// TwinCAT 3 PLC project Imbad160702PLCProgram
// ProgramVersion: 3.1.4020.4
// libraries:
//   Tc2_SerialCom, * (Beckhoff Automation GmbH)
//   Tc2_Standard, * (Beckhoff Automation GmbH)
//   Tc2_System, * (Beckhoff Automation GmbH)
//   Tc2_TcpIp, * (Beckhoff Automation GmbH)
//   Tc2_Utilities, * (Beckhoff Automation GmbH)
//   Tc3_Module, * (Beckhoff Automation GmbH)
//   Tc2_EthernetIP,newest,Beckhoff Automation GmbH
// project tree:
//   DUTs/CycleStationControl/ eAutoBaggerState.TcDUT, eCapInsertStaState.TcDUT, eGoodULStaState.TcDUT, eGoodULNewStaState.TcDUT, eVisionStaState.TcDUT, eOB_StopBeforeVisionState.TcDUT, eRejectStaState.TcDUT, ePistonInsertStaState.TcDUT, eIB_StopRobotClearStaState.TcDUT, eLoadSta1State.TcDUT, eOB_StopRobotClearStaState.TcDUT, eLoadSta2State.TcDUT, eLoadSta3State.TcDUT, eLoadSta4State.TcDUT, ePrimeMoverState.TcDUT, eCycleControlState.TcDUT, OverallStationStatus.TcDUT
//   DUTs/FrameworkDUTs/ ST_EventData.TcDUT
//   DUTs/LotDataDUTs/ eBarrelType.TcDUT, eVisionEnableState.TcDUT, LotDataType.TcDUT, StatusCounts.TcDUT
//   DUTs/Magnemotion/ eMM_HLCStatus.TcDUT, eMM_ResetCmdStatus.TcDUT, eMM_StartupCmdStatus.TcDUT, eMM_VehicleState.TcDUT, eMM_VehMoveToPosCmdStatus.TcDUT, ST_B1Cmd.TcDUT, ST_B1Res.TcDUT, ST_B2Cmd.TcDUT, ST_B2Res.TcDUT, ST_B3Cmd.TcDUT, ST_B3Res.TcDUT, ST_B4Cmd.TcDUT, ST_B4Res.TcDUT, ST_B5Cmd.TcDUT, ST_B8Cmd.TcDUT, ST_B8Res.TcDUT, ST_MM_Header.TcDUT, ST_MM_ResDataNamed.TcDUT, ST_MM_ResHeader.TcDUT, ST_MM_RxFrame.TcDUT, ST_MM_TxFrame.TcDUT, ST_ResD0.TcDUT, ST_ResD1.TcDUT, ST_ResD2.TcDUT, ST_ResD3.TcDUT, ST_ResD4.TcDUT, ST_ResD5.TcDUT, ST_ResD7.TcDUT, ST_VehicleStatus.TcDUT, ST_VehicleStatusHMI.TcDUT, U_MM_CmdData.TcDUT, U_MM_ResCmdDataDetail.TcDUT, U_MM_ResD0CmdDataDetail.TcDUT, U_MM_ResData.TcDUT
//   DUTs/PartsDataDUTs/ ePartStatus.TcDUT, PartDataType.TcDUT, VisionInspectDataType.TcDUT
//   GVLs/ CONFIG.TcGVL, GVL_IO.TcGVL, Logging.TcGVL, LotsData.TcGVL, MM_CONST.TcGVL, PartsData.TcGVL, Stations.TcGVL, STATUS.TcGVL, VIS_CONST.TcGVL
//   / PlcTask.TcTTO, SerialComTask.TcTTO
//   POUs/ AutoBagger.TcPOU, BurnOffStation.TcPOU, CapInsertStation.TcPOU, CapInsertStation_Old.TcPOU, CheckBounds.TcPOU, CycleControl.TcPOU, GoodULStation_2.TcPOU, GoodULStation_3.TcPOU, GoodULStation_4.TcPOU, GoodUnloadStation.TcPOU, IB_StopRobotClearStation.TcPOU, Load1Station.TcPOU, Load2Station.TcPOU, Load3Station.TcPOU, Load4Station.TcPOU, OB_StopRobotClearStation.TcPOU, PistonInsertStation.TcPOU, PrimeMover.TcPOU, MAIN.TcPOU, P_TextModeWrite.TcPOU, P_TextModeWriteLot.TcPOU, RejectStation.TcPOU, GoodULStation_1.TcPOU, RoutePlanner.TcPOU, StationManager.TcPOU, OB_StopBeforeVisionStation.TcPOU, VehicleManager.TcPOU, VisionStation.TcPOU
//   POUs/FrameworkPOUs/ BackgroundEL.TcPOU, EventMsg.TcPOU, EventMsgParams.TcPOU, FB_SerialCom.TcPOU, LotLogging.TcPOU, GetInputsFromFieldBus.TcPOU, MapLockedOutputsfromHMI.TcPOU, PrepareInputsDataStructureForHMI.TcPOU, PrepareOutputsDataStructureForHMI.TcPOU, SetOutputsToFieldBus.TcPOU
//   POUs/MagneMotion/HelperPOUs/ FB_LogFifo.TcPOU, FB_Rx_FrameFifo.TcPOU, FB_Tx_FrameFifo.TcPOU, F_ADSLOGHEXDATA.TcPOU
//   POUs/MagneMotion/ HLCConnection.TcPOU, MMClient.TcPOU, MMStatusMonitor.TcPOU, MM_MsgFormatter.TcPOU, MM_MsgParser.TcPOU
// real-time tasks:
//   TASK PlcTask: cycle T#10ms, priority 20, ADS port 350
//   TASK SerialComTask: cycle T#1ms, priority 16, ADS port 351
// I/O:
//   DEVICE Device 1 (EtherCAT), AmsNetId 5.37.254.56.2.1
//     Term 1 (EK1200) [EK1200-5000 EtherCAT Power supply (2A E-Bus)]
//       Term 2 (EL1809) [EL1809 16Ch. Dig. Input 24V, 3ms]
//       Term 3 (EL1088) [EL1088 8Ch. Dig. Input 24V, 3ms, negative]
//       Term 4 (EL2809) [EL2809 16Ch. Dig. Output 24V, 0.5A]
//       Term 5 (EL3312) [EL3312 2Ch. Ana. Input Thermocouple (TC)]
//       Term 6 (EL4002) [EL4002 2Ch. Ana. Output 0-10V, 12bit]
//       Term 7 (EL6001) [EL6001 Interface (RS232)]
//       Term 20 (EL2624) [EL2624 4Ch. Relay Output, NO (125V AC / 30V DC)]
//       Term 25 (EL2084) [EL2084 4Ch. Dig. Output 24V, 0.5A, switching to negative]
//       Term 10 (EK1122) [EK1122 2 port EtherCAT junction]
//         Box 37 (EP1809-0021) [EP1809-0021 16 Ch. Dig. Input 24V, 3ms, M8]
//         Box 24 (EX260-SEC1) [EX260-SEC1 EtherCAT SI Unit (32DO_PNP) Rev1.2]
//         Box 41 (EP2339-0021) [EP2339-0021 16 Ch. Dig. Input/Output 24V, 0,5A, M8]
//         Box 42 (EP1809-0021) [EP1809-0021 16 Ch. Dig. Input 24V, 3ms, M8]
//         Box 43 (EP1809-0021) [EP1809-0021 16 Ch. Dig. Input 24V, 3ms, M8]
//         Box 11 (EX260-SEC1) [EX260-SEC1 EtherCAT SI Unit (32DO_PNP) Rev1.2]
//         Box 32 (JXCE1) [JXCE1 EtherCAT JXC Rev.1.1]
//   DEVICE Device 2 (TC3 EIP Scanner), AmsNetId 5.55.113.178.3.1
//     CV-X400 Series // <INFO> 192.168.0.31, CV-X400 Series (ProdCode: 5005, Rev: 1.01, Mac: 00:01:fc:21:1c:0d) </INFO> <EDS> </EDS>
// variable links:
//   Imbad160702PLCProgram/Imbad160702PLCProgram Instance <-> Device 1 (EtherCAT)/Term 1 (EK1200)/Term 10 (EK1122)/Box 11 (EX260-SEC1)
//     PlcTask Outputs/GVL_IO.SMCEX260_2_Byte{0..3} <-> Byte {0..3}/Output  (4 links)
//   Imbad160702PLCProgram/Imbad160702PLCProgram Instance <-> Device 1 (EtherCAT)/Term 1 (EK1200)/Term 10 (EK1122)/Box 24 (EX260-SEC1)
//     PlcTask Outputs/GVL_IO.SMCEX260_1_Byte{0..3} <-> Byte {0..3}/Output  (4 links)
//   Imbad160702PLCProgram/Imbad160702PLCProgram Instance <-> Device 1 (EtherCAT)/Term 1 (EK1200)/Term 10 (EK1122)/Box 32 (JXCE1)
//     PlcTask Inputs/GVL_IO.SMC_LEY_XCurrMtrPos <-> Tx PDO1 Mapping/Current position
//     PlcTask Inputs/GVL_IO.SMC_LEY_XUINT0 <-> Tx PDO1 Mapping/Signal allocated to the input port
//     PlcTask Inputs/GVL_IO.SMC_LEY_XUINT1 <-> Tx PDO1 Mapping/Controller information flag
//     PlcTask Outputs/GVL_IO.SMC_LEY_YUINT0 <-> Rx PDO1 Mapping/Output port to which signals are allcated
//   Imbad160702PLCProgram/Imbad160702PLCProgram Instance <-> Device 1 (EtherCAT)/Term 1 (EK1200)/Term 10 (EK1122)/Box 37 (EP1809-0021)
//     PlcTask Inputs/GVL_IO.LD_XPalletCloseExtended_1_2 <-> Channel 2/Input
//     PlcTask Inputs/GVL_IO.LD_XPalletCloseExtended_3_4 <-> Channel 4/Input
//     PlcTask Inputs/GVL_IO.LD_XPalletCloseRetracted_1_2 <-> Channel 1/Input
//     PlcTask Inputs/GVL_IO.LD_XPalletCloseRetracted_3_4 <-> Channel 3/Input
//     PlcTask Inputs/GVL_IO.LD_XPalletHoldDownExtendHome <-> Channel 14/Input
//     PlcTask Inputs/GVL_IO.LD_XPalletHoldRetractEngage <-> Channel 13/Input
//     PlcTask Inputs/GVL_IO.LD_XPalletReleaseExtended <-> Channel 16/Input
//     PlcTask Inputs/GVL_IO.LD_XPalletReleaseHome <-> Channel 15/Input
//     PlcTask Inputs/GVL_IO.PI_XEscapementAtBowl <-> Channel 7/Input
//     PlcTask Inputs/GVL_IO.PI_XEscapementAtInsertLoc <-> Channel 6/Input
//     PlcTask Inputs/GVL_IO.PI_XPalletHoldDownExtended <-> Channel 11/Input
//     PlcTask Inputs/GVL_IO.PI_XPalletHoldDownHome <-> Channel 10/Input
//     PlcTask Inputs/GVL_IO.PI_XPistonPresentEscapement <-> Channel 12/Input
//   Imbad160702PLCProgram/Imbad160702PLCProgram Instance <-> Device 1 (EtherCAT)/Term 1 (EK1200)/Term 10 (EK1122)/Box 41 (EP2339-0021)
//     PlcTask Inputs/GVL_IO.MC_XAirPressureOK <-> Channel 13/Input
//     PlcTask Inputs/GVL_IO.RJ_XPartPresent <-> Channel 16/Input
//     PlcTask Inputs/GVL_IO.UL_1_XBarrelPresent <-> Channel 11/Input
//     PlcTask Inputs/GVL_IO.UL_2_XBarrelPresent <-> Channel 12/Input
//     PlcTask Inputs/GVL_IO.UL_3_XBarrelPresent <-> Channel 14/Input
//     PlcTask Inputs/GVL_IO.UL_4_XBarrelPresent <-> Channel 15/Input
//     PlcTask Inputs/GVL_IO.YU_XLocBit0 <-> Channel 3/Input
//     PlcTask Inputs/GVL_IO.YU_XLocBit1 <-> Channel 4/Input
//     PlcTask Inputs/GVL_IO.YU_XPrepareToLoad <-> Channel 1/Input
//     PlcTask Inputs/GVL_IO.YU_XToolDown <-> Channel 5/Input
//     PlcTask Inputs/GVL_IO.YU_XToolUp <-> Channel 2/Input
//     PlcTask Outputs/GVL_IO.YU_YAckPartsHeld <-> Channel 24/Output
//     PlcTask Outputs/GVL_IO.YU_YIMBADIsOK <-> Channel 22/Output
//     PlcTask Outputs/GVL_IO.YU_YOkToLoad <-> Channel 23/Output
//   Imbad160702PLCProgram/Imbad160702PLCProgram Instance <-> Device 1 (EtherCAT)/Term 1 (EK1200)/Term 10 (EK1122)/Box 42 (EP1809-0021)
//     PlcTask Inputs/GVL_IO.BG_XChute1Closed <-> Channel 14/Input
//     PlcTask Inputs/GVL_IO.BG_XChute2Closed <-> Channel 8/Input
//     PlcTask Inputs/GVL_IO.BG_XChute3Closed <-> Channel 11/Input
//     PlcTask Inputs/GVL_IO.BG_XChute4Closed <-> Channel 12/Input
//     PlcTask Inputs/GVL_IO.BG_XChute1Open <-> Channel 7/Input
//     PlcTask Inputs/GVL_IO.BG_XChute2Open <-> Channel 9/Input
//     PlcTask Inputs/GVL_IO.BG_XChute3Open <-> Channel 10/Input
//     PlcTask Inputs/GVL_IO.BG_XChute4Open <-> Channel 13/Input
//     PlcTask Inputs/GVL_IO.RJ_XPalletHoldDownExtended_Home <-> Channel 4/Input
//     PlcTask Inputs/GVL_IO.RJ_XPalletHoldDownRetracted_Engaged <-> Channel 5/Input
//     PlcTask Inputs/GVL_IO.UL_3_XPalletHoldDownRetracted_Engaged <-> Channel 1/Input
//     PlcTask Inputs/GVL_IO.UL_4_XPalletHoldDownRetracted_Engaged <-> Channel 3/Input
//     PlcTask Inputs/GVL_IO.UL_4_XPalletHoldDownExtended_Home <-> Channel 2/Input
//   Imbad160702PLCProgram/Imbad160702PLCProgram Instance <-> Device 1 (EtherCAT)/Term 1 (EK1200)/Term 10 (EK1122)/Box 43 (EP1809-0021)
//     PlcTask Inputs/GVL_IO.CP_XCapSlideExtended <-> Channel 5/Input
//     PlcTask Inputs/GVL_IO.CP_XCapSlideRetracted <-> Channel 6/Input
//     PlcTask Inputs/GVL_IO.CP_XPalletHoldDownExtended <-> Channel 2/Input
//     PlcTask Inputs/GVL_IO.CP_XPalletHoldDownHome <-> Channel 1/Input
//     PlcTask Inputs/GVL_IO.UL_1_XPalletHoldDownExtended_Home <-> Channel 12/Input
//     PlcTask Inputs/GVL_IO.UL_2_XPalletHoldDownExtended_Home <-> Channel 14/Input
//     PlcTask Inputs/GVL_IO.UL_3_XPalletHoldDownExtended_Home <-> Channel 16/Input
//     PlcTask Inputs/GVL_IO.UL_1_XPalletHoldDownRetracted_Engaged <-> Channel 13/Input
//     PlcTask Inputs/GVL_IO.UL_2_XPalletHoldDownRetracted_Engaged <-> Channel 15/Input
//   Imbad160702PLCProgram/Imbad160702PLCProgram Instance <-> Device 1 (EtherCAT)/Term 1 (EK1200)/Term 2 (EL1809)
//     PlcTask Inputs/GVL_IO.BG_XBaggerOKNoFault <-> Channel 12/Input
//     PlcTask Inputs/GVL_IO.BG_XBaggerReadyForFiller <-> Channel 14/Input
//     PlcTask Inputs/GVL_IO.BG_XBaggerWaitingForLabel <-> Channel 13/Input
//     PlcTask Inputs/GVL_IO.BG_XBagsLow <-> Channel 11/Input
//     PlcTask Inputs/GVL_IO.BU_XAlarm <-> Channel 1/Input
//     PlcTask Inputs/GVL_IO.MC_NotEStopped <-> Channel 7/Input
//     PlcTask Inputs/GVL_IO.MC_XStartPB <-> Channel 3/Input
//     PlcTask Inputs/GVL_IO.MC_XStopPB <-> Channel 4/Input
//   Imbad160702PLCProgram/Imbad160702PLCProgram Instance <-> Device 1 (EtherCAT)/Term 1 (EK1200)/Term 20 (EL2624)
//     PlcTask Outputs/GVL_IO.BG_YFillerTrigger <-> Channel 2/Output
//     PlcTask Outputs/GVL_IO.IZ_YInterrupt <-> Channel 3/Output
//     PlcTask Outputs/GVL_IO.MM_YEnableMagneMotion <-> Channel 1/Output
//   Imbad160702PLCProgram/Imbad160702PLCProgram Instance <-> Device 1 (EtherCAT)/Term 1 (EK1200)/Term 3 (EL1088)
//     PlcTask Inputs/GVL_IO.BG_XBaggerBusy <-> Channel 4/Input
//     PlcTask Inputs/GVL_IO.IZ_XAlarm <-> Channel 3/Input
//     PlcTask Inputs/GVL_IO.IZ_XConditionAlarm <-> Channel 2/Input
//     PlcTask Inputs/GVL_IO.IZ_XIonAlarm <-> Channel 1/Input
//   Imbad160702PLCProgram/Imbad160702PLCProgram Instance <-> Device 1 (EtherCAT)/Term 1 (EK1200)/Term 4 (EL2809)
//     PlcTask Outputs/GVL_IO.MC_YStackLightGreen <-> Channel 15/Output
//     PlcTask Outputs/GVL_IO.MC_YStackLightRed <-> Channel 13/Output
//     PlcTask Outputs/GVL_IO.MC_YStackLightYellow <-> Channel 14/Output
//     PlcTask Outputs/GVL_IO.VS_YBarrelLED_off <-> Channel 12/Output
//   Imbad160702PLCProgram/Imbad160702PLCProgram Instance <-> Device 1 (EtherCAT)/Term 1 (EK1200)/Term 5 (EL3312)
//     PlcTask Inputs/GVL_IO.BU_Temperature <-> TC Inputs Channel 1/Value
//   Imbad160702PLCProgram/Imbad160702PLCProgram Instance <-> Device 1 (EtherCAT)/Term 1 (EK1200)/Term 6 (EL4002)
//     PlcTask Outputs/GVL_IO.BU_BlowCntl <-> AO Outputs Channel 2/Analog output
//     PlcTask Outputs/GVL_IO.BU_HeatCntl <-> AO Outputs Channel 1/Analog output
//   Imbad160702PLCProgram/Imbad160702PLCProgram Instance <-> Device 1 (EtherCAT)/Term 1 (EK1200)/Term 7 (EL6001)
//     SerialComTask Inputs/BackgroundEL.stIn_EL6001/D <-> COM Inputs/Data In 0
//     SerialComTask Inputs/BackgroundEL.stIn_EL6001/D @bit {8..168 step 8} <-> COM Inputs/Data In {1..21}  (21 links)
//     SerialComTask Inputs/BackgroundEL.stIn_EL6001/Status <-> COM Inputs/Status
//     SerialComTask Outputs/BackgroundEL.stOut_EL6001/Ctrl <-> COM Outputs/Ctrl
//     SerialComTask Outputs/BackgroundEL.stOut_EL6001/D <-> COM Outputs/Data Out 0
//     SerialComTask Outputs/BackgroundEL.stOut_EL6001/D @bit {8..168 step 8} <-> COM Outputs/Data Out {1..21}  (21 links)
//   Imbad160702PLCProgram/Imbad160702PLCProgram Instance <-> Device 2 (TC3 EIP Scanner)/CV-X400 Series
//     PlcTask Inputs/GVL_IO.VS_XByte0 <-> Connection 1 (Input/Output)/Inputs/InByte
//     PlcTask Inputs/GVL_IO.VS_XByte1 <-> Connection 1 (Input/Output)/Inputs/InByte_2
//     PlcTask Inputs/GVL_IO.VS_XByte100 <-> Connection 1 (Input/Output)/Inputs/InByte_101
//     PlcTask Inputs/GVL_IO.VS_XByte101 <-> Connection 1 (Input/Output)/Inputs/InByte_102
//     PlcTask Inputs/GVL_IO.VS_XByte102 <-> Connection 1 (Input/Output)/Inputs/InByte_103
//     PlcTask Inputs/GVL_IO.VS_XByte103 <-> Connection 1 (Input/Output)/Inputs/InByte_104
//     PlcTask Inputs/GVL_IO.VS_XByte108 <-> Connection 1 (Input/Output)/Inputs/InByte_109
//     PlcTask Inputs/GVL_IO.VS_XByte109 <-> Connection 1 (Input/Output)/Inputs/InByte_110
//     PlcTask Inputs/GVL_IO.VS_XByte110 <-> Connection 1 (Input/Output)/Inputs/InByte_111
//     PlcTask Inputs/GVL_IO.VS_XByte111 <-> Connection 1 (Input/Output)/Inputs/InByte_112
//     PlcTask Inputs/GVL_IO.VS_XByte112 <-> Connection 1 (Input/Output)/Inputs/InByte_113
//     PlcTask Inputs/GVL_IO.VS_XByte113 <-> Connection 1 (Input/Output)/Inputs/InByte_114
//     PlcTask Inputs/GVL_IO.VS_XByte114 <-> Connection 1 (Input/Output)/Inputs/InByte_115
//     PlcTask Inputs/GVL_IO.VS_XByte115 <-> Connection 1 (Input/Output)/Inputs/InByte_116
//     PlcTask Inputs/GVL_IO.VS_XByte116 <-> Connection 1 (Input/Output)/Inputs/InByte_117
//     PlcTask Inputs/GVL_IO.VS_XByte117 <-> Connection 1 (Input/Output)/Inputs/InByte_118
//     PlcTask Inputs/GVL_IO.VS_XByte118 <-> Connection 1 (Input/Output)/Inputs/InByte_119
//     PlcTask Inputs/GVL_IO.VS_XByte119 <-> Connection 1 (Input/Output)/Inputs/InByte_120
//     PlcTask Inputs/GVL_IO.VS_XByte120 <-> Connection 1 (Input/Output)/Inputs/InByte_121
//     PlcTask Inputs/GVL_IO.VS_XByte121 <-> Connection 1 (Input/Output)/Inputs/InByte_122
//     PlcTask Inputs/GVL_IO.VS_XByte122 <-> Connection 1 (Input/Output)/Inputs/InByte_123
//     PlcTask Inputs/GVL_IO.VS_XByte123 <-> Connection 1 (Input/Output)/Inputs/InByte_124
//     PlcTask Inputs/GVL_IO.VS_XByte2 <-> Connection 1 (Input/Output)/Inputs/InByte_3
//     PlcTask Inputs/GVL_IO.VS_XByte20 <-> Connection 1 (Input/Output)/Inputs/InByte_21
//     PlcTask Inputs/GVL_IO.VS_XByte24 <-> Connection 1 (Input/Output)/Inputs/InByte_25
//     PlcTask Inputs/GVL_IO.VS_XByte28 <-> Connection 1 (Input/Output)/Inputs/InByte_29
//     PlcTask Inputs/GVL_IO.VS_XByte3 <-> Connection 1 (Input/Output)/Inputs/InByte_4
//     PlcTask Inputs/GVL_IO.VS_XByte4 <-> Connection 1 (Input/Output)/Inputs/InByte_5
//     PlcTask Inputs/GVL_IO.VS_XByte48 <-> Connection 1 (Input/Output)/Inputs/InByte_49
//     PlcTask Inputs/GVL_IO.VS_XByte49 <-> Connection 1 (Input/Output)/Inputs/InByte_50
//     PlcTask Inputs/GVL_IO.VS_XByte50 <-> Connection 1 (Input/Output)/Inputs/InByte_51
//     PlcTask Inputs/GVL_IO.VS_XByte51 <-> Connection 1 (Input/Output)/Inputs/InByte_52
//     PlcTask Inputs/GVL_IO.VS_XByte52 <-> Connection 1 (Input/Output)/Inputs/InByte_53
//     PlcTask Inputs/GVL_IO.VS_XByte53 <-> Connection 1 (Input/Output)/Inputs/InByte_54
//     PlcTask Inputs/GVL_IO.VS_XByte54 <-> Connection 1 (Input/Output)/Inputs/InByte_55
//     PlcTask Inputs/GVL_IO.VS_XByte55 <-> Connection 1 (Input/Output)/Inputs/InByte_56
//     PlcTask Inputs/GVL_IO.VS_XByte56 <-> Connection 1 (Input/Output)/Inputs/InByte_57
//     PlcTask Inputs/GVL_IO.VS_XByte57 <-> Connection 1 (Input/Output)/Inputs/InByte_58
//     PlcTask Inputs/GVL_IO.VS_XByte58 <-> Connection 1 (Input/Output)/Inputs/InByte_59
//     PlcTask Inputs/GVL_IO.VS_XByte59 <-> Connection 1 (Input/Output)/Inputs/InByte_60
//     PlcTask Inputs/GVL_IO.VS_XByte60 <-> Connection 1 (Input/Output)/Inputs/InByte_61
//     PlcTask Inputs/GVL_IO.VS_XByte61 <-> Connection 1 (Input/Output)/Inputs/InByte_62
//     PlcTask Inputs/GVL_IO.VS_XByte62 <-> Connection 1 (Input/Output)/Inputs/InByte_63
//     PlcTask Inputs/GVL_IO.VS_XByte63 <-> Connection 1 (Input/Output)/Inputs/InByte_64
//     PlcTask Inputs/GVL_IO.VS_XByte64 <-> Connection 1 (Input/Output)/Inputs/InByte_65
//     PlcTask Inputs/GVL_IO.VS_XByte65 <-> Connection 1 (Input/Output)/Inputs/InByte_66
//     PlcTask Inputs/GVL_IO.VS_XByte66 <-> Connection 1 (Input/Output)/Inputs/InByte_67
//     PlcTask Inputs/GVL_IO.VS_XByte67 <-> Connection 1 (Input/Output)/Inputs/InByte_68
//     PlcTask Inputs/GVL_IO.VS_XByte68 <-> Connection 1 (Input/Output)/Inputs/InByte_69
//     PlcTask Inputs/GVL_IO.VS_XByte69 <-> Connection 1 (Input/Output)/Inputs/InByte_70
//     PlcTask Inputs/GVL_IO.VS_XByte70 <-> Connection 1 (Input/Output)/Inputs/InByte_71
//     PlcTask Inputs/GVL_IO.VS_XByte71 <-> Connection 1 (Input/Output)/Inputs/InByte_72
//     PlcTask Inputs/GVL_IO.VS_XByte72 <-> Connection 1 (Input/Output)/Inputs/InByte_73
//     PlcTask Inputs/GVL_IO.VS_XByte73 <-> Connection 1 (Input/Output)/Inputs/InByte_74
//     PlcTask Inputs/GVL_IO.VS_XByte74 <-> Connection 1 (Input/Output)/Inputs/InByte_75
//     PlcTask Inputs/GVL_IO.VS_XByte75 <-> Connection 1 (Input/Output)/Inputs/InByte_76
//     PlcTask Inputs/GVL_IO.VS_XByte76 <-> Connection 1 (Input/Output)/Inputs/InByte_77
//     PlcTask Inputs/GVL_IO.VS_XByte77 <-> Connection 1 (Input/Output)/Inputs/InByte_78
//     PlcTask Inputs/GVL_IO.VS_XByte78 <-> Connection 1 (Input/Output)/Inputs/InByte_79
//     PlcTask Inputs/GVL_IO.VS_XByte79 <-> Connection 1 (Input/Output)/Inputs/InByte_80
//     PlcTask Inputs/GVL_IO.VS_XByte80 <-> Connection 1 (Input/Output)/Inputs/InByte_81
//     PlcTask Inputs/GVL_IO.VS_XByte81 <-> Connection 1 (Input/Output)/Inputs/InByte_82
//     PlcTask Inputs/GVL_IO.VS_XByte82 <-> Connection 1 (Input/Output)/Inputs/InByte_83
//     PlcTask Inputs/GVL_IO.VS_XByte83 <-> Connection 1 (Input/Output)/Inputs/InByte_84
//     PlcTask Inputs/GVL_IO.VS_XByte88 <-> Connection 1 (Input/Output)/Inputs/InByte_89
//     PlcTask Inputs/GVL_IO.VS_XByte89 <-> Connection 1 (Input/Output)/Inputs/InByte_90
//     PlcTask Inputs/GVL_IO.VS_XByte90 <-> Connection 1 (Input/Output)/Inputs/InByte_91
//     PlcTask Inputs/GVL_IO.VS_XByte91 <-> Connection 1 (Input/Output)/Inputs/InByte_92
//     PlcTask Inputs/GVL_IO.VS_XByte92 <-> Connection 1 (Input/Output)/Inputs/InByte_93
//     PlcTask Inputs/GVL_IO.VS_XByte93 <-> Connection 1 (Input/Output)/Inputs/InByte_94
//     PlcTask Inputs/GVL_IO.VS_XByte94 <-> Connection 1 (Input/Output)/Inputs/InByte_95
//     PlcTask Inputs/GVL_IO.VS_XByte95 <-> Connection 1 (Input/Output)/Inputs/InByte_96
//     PlcTask Inputs/GVL_IO.VS_XByte96 <-> Connection 1 (Input/Output)/Inputs/InByte_97
//     PlcTask Inputs/GVL_IO.VS_XByte97 <-> Connection 1 (Input/Output)/Inputs/InByte_98
//     PlcTask Inputs/GVL_IO.VS_XByte98 <-> Connection 1 (Input/Output)/Inputs/InByte_99
//     PlcTask Inputs/GVL_IO.VS_XByte99 <-> Connection 1 (Input/Output)/Inputs/InByte_100
//     PlcTask Outputs/GVL_IO.VS_YByte0 <-> Connection 1 (Input/Output)/Outputs/OutByte
//     PlcTask Outputs/GVL_IO.VS_YByte1 <-> Connection 1 (Input/Output)/Outputs/OutByte_2
//     PlcTask Outputs/GVL_IO.VS_YByte16 <-> Connection 1 (Input/Output)/Outputs/OutByte_17
//     PlcTask Outputs/GVL_IO.VS_YByte2 <-> Connection 1 (Input/Output)/Outputs/OutByte_3
//     PlcTask Outputs/GVL_IO.VS_YByte20 <-> Connection 1 (Input/Output)/Outputs/OutByte_21
//     PlcTask Outputs/GVL_IO.VS_YByte24 <-> Connection 1 (Input/Output)/Outputs/OutByte_25

CONFIGURATION Imbad160702PLCProgram
    RESOURCE PLC ON TwinCAT3
        TASK PlcTask(INTERVAL := T#10ms, PRIORITY := 20);
        TASK SerialComTask(INTERVAL := T#1ms, PRIORITY := 16);
        PROGRAM MAIN WITH PlcTask : MAIN;
        PROGRAM BackgroundEL WITH SerialComTask : BackgroundEL;
    END_RESOURCE
END_CONFIGURATION

// ---- DUTs/CycleStationControl/eAutoBaggerState.TcDUT
{attribute 'qualified_only'}
{attribute 'strict'}
TYPE eAutoBaggerState :
(
	eUnknown  :=1 ,
	
	eError,

//Init? send label delete, reset, etc?
	eInit,
	
// Check if bagger is not faulted and waiting for label	and has no low bag warning
    eCheckWaitingLabel,

//wait for one chute to fill up
	eReady,

//open trap door, selecting correct one
//wait for 2 seconds or something
	eDropParts,

	eDoorCannotOpen,
	
//then close the trap door
    eHalfCloseTrapDoor,
    
    eOpenTrapDoor,
	
	eOpenTrapDoorFinal,
	
	eCloseTrapDoor,
	
	eCloseTrapDoorFinal,
	
	eDoorCannotClose,

//send label and print command
	eSendLabel,
	
	eMissingBusySignal,
	
	eMissingBusySignal2,
	
	eMissingNotBusySignal,

//wait for bagger ready, then send feeder ready command
	eDetachBag1,
	
	eDetachBag2,
	
	eFeederReadyReset1,
	
	eFeederReadyReset2,
	
	eWaitForBaggerNotBusy,
	
	eWaitForBaggerBusy,
	
	eWaitForBagOpen,
	
	eHandleBagOpenError,
	
	eTriggerBagger,
	
	eWaitforBaggingStart,
	
	eWaitforBaggingComplete


);
END_TYPE

// ---- DUTs/CycleStationControl/eCapInsertStaState.TcDUT
{attribute 'qualified_only'}
{attribute 'strict'}
TYPE eCapInsertStaState :
( 
	eUnknown := 51,
	eHoming,
	eDisabledReady,
	eWaitForVehicleTrigger,
	ePalletHoldDownGoingDown,
	ePalletHoldDownExtended,
	eCapSlideGoingDown,
	eCapSlideExtended,
	eCapSlideGoingUp,
	eCapSlideUp,
	ePalletHoldDownGoingUp,
	ePalletHoldDownUp,
	eDepart,
	eStopActive,
    eError
);
END_TYPE

// ---- DUTs/CycleStationControl/eGoodULStaState.TcDUT
{attribute 'qualified_only'}
{attribute 'strict'}
TYPE eGoodULStaState :
( 
	eUnknown :=151,
    eInit,
	eHoming,
	eHPReset,
	eHPCheckEnabled,
	eHPSendHome,
	eHPHomed,
	eHPSendToInitLoc,
	eHPAtInitLoc,
	eHPReady,
	eDisabledReady,
    eWaitForVehicleTrigger,
	eDetermineDropLocation,
	eDwell,
	eAbandonCycle,
	eEngagePalletHoldDown,
	ePalletHoldDownEngaged,
	ePalletReleaseExtend,
	ePalletReleaseExtended,
    eWaitForHPInitLocAndRotaryCenter,	
	eHPMoveToPickFromTrack,
	eHPAtPickFromTrack,
	eHPCloseGrippers,
	eHPGrippersClosed,
	eHPSendToInitLocNext,
	eHPAtInitLocNext,
	eReleasePalletHoldDown,
	ePalletHoldDownReleased,	
	eHPMoveToPlaceInBagLoc1,
	eHPMoveToPlaceInBagLoc2,
	eHPAtPlaceinBagLoc1,
	eHPAtPlaceinBagLoc2,
	eDepartVehicle,
	eTurnToRotartyCorrectSide,
	eAtCorrectRotaryLoc,
	eHPOpenGrippers,
	eHPGrippersOpen,	
	eMoveRotaryRight,
	eCheckRotaryAtRight,		
	eHPSendToInitLocAfterDrop,	
    eHPAtInitLocAfterDrop,
	eHPMoveToRotaryCenter,
	eHPAtRotaryCenter,	
	eStopActive,
	eError
);
END_TYPE

// ---- DUTs/CycleStationControl/eGoodULNewStaState.TcDUT
{attribute 'qualified_only'}
{attribute 'strict'}
TYPE eGoodULNewStaState :
( 
	eUnknown := 701,
    eInit,
	eHoming,
	eReady,
	eDisabledReady,
	eWaitForVehicleTrigger,
	eDwell,
	eCheckChuteCount,
	eSendPalletHoldDownExtend,
	eCheckPalletHoldDownExtended,
	ePalletReleaseExtend,
	ePalletReleaseExtended,
	eKnockoffPart,
	eKnockoffExtended,
	eCheckPartKnockedOff,
	ePalletHoldDownRelease,
	ePalletHoldDownReleased,
	eDepart,
	eStopActive,
    eError
);
END_TYPE

// ---- DUTs/CycleStationControl/eVisionStaState.TcDUT
{attribute 'qualified_only'}
{attribute 'strict'}
TYPE eVisionStaState :
( 
	eUnknown := 801,
	eCheckToolPosition,
    eInit,
	eHoming,
	eCmdTriggerReset,
	eCheckTriggerResetCmpl,
	eConfirmRunState,
	eGetProgramNumber,
	eCheckProgramNumber,
	eChangeProgramNumber,
	eReady,
	eWaitingForVehicleTrigger,
	eShortShotTrigger,
	eWaitShortShotDone,
	eBarellInspectTrigger,
	eWaitBarellInspectDone,
	eProcessVisionData,
    eDepart,
	eStopActive,
    eError
);
END_TYPE

// ---- DUTs/CycleStationControl/eOB_StopBeforeVisionState.TcDUT
{attribute 'qualified_only'}
{attribute 'strict'}
TYPE eOB_StopBeforeVisionState :
( 
	eUnknown,
    eInit,
	eHoming,
	eReady,
	eDwell,
	eProcessing,
	eDepart,
	eStopActive,
    eError
);
END_TYPE

// ---- DUTs/CycleStationControl/eRejectStaState.TcDUT
{attribute 'qualified_only'}
{attribute 'strict'}
TYPE eRejectStaState :
( 
	eUnknown := 701,
    eInit,
	eHoming,
	eReady,
	eWaitForVehicleTrigger,
	eDwell,
	eSendPalletHoldDownExtend,
	eCheckPalletHoldDownExtended,
	ePalletReleaseExtend,
	ePalletReleaseExtended,
	eKnockoffPart,
	eKnockoffExtended,
	eCheckPartKnockedOff,
	ePalletHoldDownRelease,
	ePalletHoldDownReleased,
	eDepart,
	eStopActive,
    eError
);
END_TYPE

// ---- DUTs/CycleStationControl/ePistonInsertStaState.TcDUT
{attribute 'qualified_only'}
{attribute 'strict'}
TYPE ePistonInsertStaState :
( 
	eUnknown :=601 ,
	eInit,
	eHoming,
	eSMCMtrReset,
	eSMCMtrCheckEnabled,
	eSMCMtrSendHome,
	eSMCMtrHomed,
	eCheckToolPosition,
	eDisabledReady,
	eReady,
	ePalletHoldDownEngaged,
	eMoveEscapemttoBowl,
	eEscapmentAtBowl,
	eWaitForPartAtBowl,
	eMoveEscapmentToWork,
	eEscapementAtWork,
	eFirePistonUp,
	eSendBarrelBackupEngage,
	eWaitForPistonStartMovUp,
	eWaitForBarrelBackupEngaged,
	eWaitForPistonMovDoneUp,
	eFirePistonDown,
	eRetractPalletHoldDownAndBackup,
	eWaitForPistonStartMovDwn,
	eRetractPalletHoldDownAndBarrel,
	eWaitForPalletHoldDownAndBackupRetracted,
	eWaitForPistonMovDoneDown,	
	eDepart,
	eStopActive,
	eError
);
END_TYPE

// ---- DUTs/CycleStationControl/eIB_StopRobotClearStaState.TcDUT
{attribute 'qualified_only'}
{attribute 'strict'}
TYPE eIB_StopRobotClearStaState :
( 
	eUnknown :=201,
    eInit,
	eHoming,
	eReady,
	eDwell,
	eProcessing,
	eDepart,
	eStopActive,
    eError
);
END_TYPE

// ---- DUTs/CycleStationControl/eLoadSta1State.TcDUT
{attribute 'qualified_only'}
{attribute 'strict'}
TYPE eLoadSta1State :
( 
	eUnknown :=301,
    eInit,
	eHoming,
	eReady, // waiting for vehicle trigger
	eWaitForYushinPrepareLoad,
	ePalletHoldDownEngage,
	ePalletHoldDownEngaged,
	ePalletHoldDownFree,
	ePalletHoldDownFreed,
	ePalletReleaseRaise,
	ePalletReleaseRaised,
	eWaitForIBTrackClear,
	eSignalYushinOKToLoad,
	eWaitForYushinToolDown,	
	ePalletCloseExtend,
	ePalletCloseExtended,
	ePalletReleaseLower,
	ePalletReleaseLowered,
	ePalletCloseRetract,
	ePalletCloseRetracted,
	eWaitForYushinToolUp,	
	eProcessing,
	eDepart,
	eStopActive,
    eError
);
END_TYPE

// ---- DUTs/CycleStationControl/eOB_StopRobotClearStaState.TcDUT
{attribute 'qualified_only'}
{attribute 'strict'}
TYPE eOB_StopRobotClearStaState :
( 
	eUnknown := 551,
    eInit,
	eHoming,
	eReady,
	eDwell,
	eProcessing,
	eDepart,
	eStopActive,
    eError
);
END_TYPE

// ---- DUTs/CycleStationControl/eLoadSta2State.TcDUT
{attribute 'qualified_only'}
{attribute 'strict'}
TYPE eLoadSta2State :
( 
	eUnknown :=351,
    eInit,
	eHoming,
	eReady,
	eDwell,
	eWaitForLoadComplete,
	eProcessing,
	eDepart,
	eStopActive,
    eError
);
END_TYPE

// ---- DUTs/CycleStationControl/eLoadSta3State.TcDUT
{attribute 'qualified_only'}
{attribute 'strict'}
TYPE eLoadSta3State :
( 
	eUnknown :=401,
    eInit,
	eHoming,
	eReady,
	eDwell,
	eWaitForLoadComplete,
	eProcessing,
	eDepart,
	eStopActive,
    eError
);
END_TYPE

// ---- DUTs/CycleStationControl/eLoadSta4State.TcDUT
{attribute 'qualified_only'}
{attribute 'strict'}
TYPE eLoadSta4State :
( 
	eUnknown :=451,
    eInit,
	eHoming,
	eReady,
	eDwell,
	eWaitForLoadComplete,
	eProcessing,
	eDepart,
	eStopActive,
    eError
);
END_TYPE

// ---- DUTs/CycleStationControl/ePrimeMoverState.TcDUT
{attribute 'qualified_only'}
{attribute 'strict'}
TYPE ePrimeMoverState :
(
	eMMUnknown :=651,
    eMMConnect,
	eMMCheckStatus,
	eMMSendResetCmd,
	eMMWaitAccceptResetCmd,
	eMMWaitCmplResetCmd,
	eMMSendStartupCmd,
	eMMWaitAcceptStartupCmd,
	eMMWaitCmplStartupCmd,
	eMMWaitCycleControlTrigger,
	eMMSendAllVehiclesToInitPosCmd,
	eMMWaitCmplAllVehiclesAtInitPos,
	eMMReadyAutoRun,
	eMMSuspendMovement,
	eMMESTOP,
	eMMResumeMovement,
	eStopActive,
	eMMError
);
END_TYPE

// ---- DUTs/CycleStationControl/eCycleControlState.TcDUT
{attribute 'qualified_only'}
{attribute 'strict'}
TYPE eCycleControlState :
(
	eUnknown := 101,
    eInit,
	eWaitForHoming,
	eReady,
	eAutoRun,
	eStartStop,
	eWaitForHomingAfterEStop,
    eError
);
END_TYPE

// ---- DUTs/CycleStationControl/OverallStationStatus.TcDUT
{attribute 'qualified_only'}
{attribute 'strict'}
TYPE OverallStationStatus :
(
	eDisabled :=0, // Gsilver
	eWarning,     //  Yellow 
	eError,       // Red  
	eHoming,      // Orange
	eWaitingForParts, // Blue
	eRunning, // Green 
	eCycleStop // Purple
);
END_TYPE

// ---- DUTs/FrameworkDUTs/ST_EventData.TcDUT
TYPE ST_EventData :
STRUCT
	


	rVal 	: LREAL;
	iVal	: UDINT;


END_STRUCT
END_TYPE

// ---- DUTs/LotDataDUTs/eBarrelType.TcDUT
{attribute 'qualified_only'}
{attribute 'strict'}
TYPE eBarrelType :
(
	Size55cc :=0,
	Size30cc,
	Size10cc,
	Size5cc,
	Size3cc
);
END_TYPE

// ---- DUTs/LotDataDUTs/eVisionEnableState.TcDUT
{attribute 'qualified_only'}
{attribute 'strict'}
TYPE eVisionEnableState :
(	
	Disabled :=0,
	Enabled,
	DataCollectOnly
);
END_TYPE

// ---- DUTs/LotDataDUTs/LotDataType.TcDUT
TYPE LotDataType :
STRUCT
	// Coming from HMI 
	PartNumber : STRING :='PartNumb';  
	PartDescription: STRING :='55ccBarrel';
	LotNumber: STRING :='LotNumb';
	JobNumber: STRING := 'JobNumb';
	LotDate: STRING :='DATE';
	PistonPartNumber : STRING :='PistonPartNumb';
	PistonLotNumber : STRING :='PistonLotNumb';
	CapPartNumber : STRING :='CapPartNumb';
	CapLotNumber : STRING :='CapLotNumb';
	RawMaterialLotNumber: STRING := 'RawLotNumb';
	Comment: STRING :='Defaults'; // Limit to 80 characters	from HMI
	BlackConPartNumber : STRING :='Black'; 
	
	AutoBaggerEnabled : BOOL := TRUE;
	QuantityInBag : BYTE := 50;
	BarrelSize: eBarrelType := eBarrelType.Size3cc; //55cc:=0, 30cc:= 1, 10cc: = 2, 5cc: = 3, 3cc: = 4
	BarrelSizeInt : DINT;
	BurnOffEnabled : BOOL := TRUE;
    BurnOffTemp : REAL := 50;
	CapInsertEnabled: BOOL := TRUE;
	CapTorqueSetPoint : REAL := 100;
	GoodUnloadEnabled : BOOL := TRUE;
	IonizerEnabled: BOOL := TRUE;
	LoadStationEnabled: BOOL := TRUE;
	PistonInsertEnabled : BOOL := TRUE;
	LotInProgress: BOOL := TRUE;
	
	PistonStroke : REAL:= 200;
	RejectUnloadEnabled : BOOL := TRUE;
	VisionStationRunSelectInt: DINT :=1;
	VisionStationRunSelect : eVisionEnableState := eVisionEnableState.DataCollectOnly; // Enabled:=1, Disabled:=0, Data Collect Only :=2
	ShortShotMinRadius: REAL := 80;//premium max individual stain area
	ShortShotMaxRadius: REAL := 80;//good max individual stain area
	TotalStainAreaMaxPremium : REAL :=100;
	TotalStainCountMaxPremium : REAL := 5;
	TotalStainAreaMaxGood: REAL := 300;
	TotalStainCountMaxGood : REAL := 20;
	IndividualStainAreaMaxPremium : REAL := 80;
	IndividualStainAreaMaxGood : REAL := 80;
	VisionProgramNumber : DINT := 1;
	ResetModeEnabled: BOOL := FALSE;
	
	
	
	// This is maintained by the machine
    LotStartTime: TIME;
	CavityCounts : ARRAY[1..CONFIG.MAX_CAVITY] OF StatusCounts;
	PLCVersion : STRING;
	
END_STRUCT
END_TYPE

// ---- DUTs/LotDataDUTs/StatusCounts.TcDUT
TYPE StatusCounts :
STRUCT
	PremiumCount: DINT;
	GoodCount: DINT;
	BadCount: DINT;
	TotalCount : DINT; //can be also obtained from the above, but keeping it for ease of use
END_STRUCT
END_TYPE

// ---- DUTs/Magnemotion/eMM_HLCStatus.TcDUT
{attribute 'qualified_only'}
{attribute 'strict'}
TYPE eMM_HLCStatus :
(
	eHLC_STATE_INIT			:=16#1,
	eHLC_STATE_DEGRADED		:=16#2,
	eHLC_STATE_OPERATIONAL	:=16#3
);
END_TYPE

// ---- DUTs/Magnemotion/eMM_ResetCmdStatus.TcDUT
{attribute 'qualified_only'}
{attribute 'strict'}
TYPE eMM_ResetCmdStatus :
(
	eMM_ResetCmdSent,
	eMM_ResetCmdAck,
	eMM_ResetCmdRejected,
	eMM_ResetCmdComplete
);
END_TYPE

// ---- DUTs/Magnemotion/eMM_StartupCmdStatus.TcDUT
{attribute 'qualified_only'}
{attribute 'strict'}
TYPE eMM_StartupCmdStatus :
(
	eMM_StartupCmdSent,
	eMM_StartupCmdAck,
	eMM_StartupCmdRejected,
	eMM_StartupCmdComplete
);
END_TYPE

// ---- DUTs/Magnemotion/eMM_VehicleState.TcDUT
{attribute 'qualified_only'}
{attribute 'strict'}
TYPE eMM_VehicleState :
(
	eVehIdle,
	eVehMoveCmd_Send,
	eVehMoveCmd_WaitAccept,
	eVehMoveCmd_Reject,
	eVehMoveCmd_WaitCompl,
	eVehMoveCmd_Compl,
	eVehMoveTimeOut,	
	eError
);
END_TYPE

// ---- DUTs/Magnemotion/eMM_VehMoveToPosCmdStatus.TcDUT
{attribute 'qualified_only'}
{attribute 'strict'}
TYPE eMM_VehMoveToPosCmdStatus :
(
	eMM_VehMoveToPosCmdSent,
	eMM_VehMoveToPosCmdAck,
	eMM_VehMoveToPosCmdRejected,
	eMM_VehMoveToPosCmdComplete
);
END_TYPE

// ---- DUTs/Magnemotion/ST_B1Cmd.TcDUT
(* B1 = Move Vehicle to Position *)
TYPE ST_B1Cmd :
STRUCT
	Cmd_Header	:BYTE	:=16#B1;	(* 1 byte*)
	OrderNumb	:UDINT	:=0;		(* 4 bytes*)
	VehicleID	:UINT	:=0;		(* 2 bytes*)
	Flags		:BYTE	:=0;		(* 1 bytes*)
	Position	:REAL	:=0.0;     (* 4 bytes*)
	PathID		:UINT	:=0; 		(*2 bytes*)
	Accn		:REAL	:=0.0; 		(* 4 bytes*)
	Velocity	:REAL	:=0.0; 		(*4 bytes*)
	FollowID	:UINT	:=0; 		(*2 bytes *) 
	CRC			:UINT   :=0;        (*2 bytes *) 
    //CRC1		:BYTE	:=16#00;    (* 1 byte*)
	//CRC2		:BYTE	:=16#00;    (* 2 byte*)
	
END_STRUCT
END_TYPE

// ---- DUTs/Magnemotion/ST_B1Res.TcDUT
(* B1 = Move Vehicle to Position *)
TYPE ST_B1Res :
STRUCT
	OrderNumb		:UDINT;		(* 4 bytes*)
	VehicleID		:UINT;		(* 2 bytes*)	
	Position		:REAL;	    (* 4 bytes*)
	PathID			:UINT;		(*2 bytes*)
	AccnLimit		:REAL;		(* 4 bytes*)
	VelocityLimit	:REAL;		(*4 bytes*)
	Flags			:BYTE;      (*1 byte*)
	(*FollowID	    :UINT*)	    (*2 bytes *) 
	CRC1			:BYTE;	    (* 1 byte*)
	CRC2			:BYTE;	    (* 1 byte*)	
END_STRUCT
END_TYPE

// ---- DUTs/Magnemotion/ST_B2Cmd.TcDUT
(* B2 = Statrup *)
TYPE ST_B2Cmd :
STRUCT
	Cmd_Header	:BYTE	:=16#B2;	(* 1 byte*)
	PathID		:UINT	:=0; 		(* 2 bytes*)
	CRC			:UINT   :=0;        (*2 bytes *) 
	//CRC1		:BYTE	:=16#00;    (* 1 byte*)
	//CRC2		:BYTE	:=16#00;    (* 1 byte*)
	
END_STRUCT
END_TYPE

// ---- DUTs/Magnemotion/ST_B2Res.TcDUT
(* B2 = Statrup *)
TYPE ST_B2Res :
STRUCT
	PathID			:UINT;		(* 2 bytes*)
	CRC1			:BYTE;	    (* 1 byte*)
	CRC2			:BYTE;	    (* 1 byte*)	
END_STRUCT
END_TYPE

// ---- DUTs/Magnemotion/ST_B3Cmd.TcDUT
(* B3 = Resume Movement *)
TYPE ST_B3Cmd :
STRUCT
	Cmd_Header	:BYTE	:=16#B3;	(* 1 byte*)
	PathID		:UINT	:=0; 		(*2 bytes*)
	CRC			:UINT   :=0;        (*2 bytes *) 	 
	//CRC1		:BYTE	:=16#00;    (* 1 byte*)
	//CRC2		:BYTE	:=16#00;    (* 2 byte*)
	
END_STRUCT
END_TYPE

// ---- DUTs/Magnemotion/ST_B3Res.TcDUT
(* B3 = Resume Movement *)
TYPE ST_B3Res :
STRUCT
	PathID			:UINT;		(* 2 bytes*)
	CRC1			:BYTE;	    (* 1 byte*)
	CRC2			:BYTE;	    (* 1 byte*)		
END_STRUCT
END_TYPE

// ---- DUTs/Magnemotion/ST_B4Cmd.TcDUT
(* B4 = Suspend Movement *)
TYPE ST_B4Cmd :
STRUCT
	Cmd_Header	:BYTE	:=16#B4;	(* 1 byte*)
	PathID		:UINT	:=0; 		(*2 bytes*)
	CRC			:UINT   :=0;        (*2 bytes *) 
	//CRC1		:BYTE	:=16#00;    (* 1 byte*)
	//CRC2		:BYTE	:=16#00;    (* 2 byte*)
	
END_STRUCT
END_TYPE

// ---- DUTs/Magnemotion/ST_B4Res.TcDUT
(* B4 = Suspend Movement *)
TYPE ST_B4Res :
STRUCT
	PathID			:UINT;		(* 2 bytes*)
	CRC1			:BYTE;	    (* 1 byte*)
	CRC2			:BYTE;	    (* 1 byte*)		
	
END_STRUCT
END_TYPE

// ---- DUTs/Magnemotion/ST_B5Cmd.TcDUT
(* B5 = Status Request *)
TYPE ST_B5Cmd :
STRUCT
	//Cmd_Header	:BYTE	:=16#B5;	(* 1 byte*)
	ReqType		:BYTE	:=0;		(* 1 bytes*)
	ID			:UINT	:=0;		(* 2 bytes*)
	MotorIndex	:BYTE	:=0;		(* 1 bytes*)
	CRC			:UINT   :=0;        (*2 bytes *) 
    //CRC1		:BYTE	:=16#00;    (* 1 byte*)
	//CRC2		:BYTE	:=16#00;    (* 2 byte*)
	
END_STRUCT
END_TYPE

// ---- DUTs/Magnemotion/ST_B8Cmd.TcDUT
(* B8 = Reset *)
TYPE ST_B8Cmd :
STRUCT
	PathID		:UINT	:=0; 		(* 2 bytes*)
	CRC			:UINT   :=0;        (*2 bytes *)     
    //CRC1		:BYTE	:=16#00;    (* 1 byte*)
	//CRC2		:BYTE	:=16#00;    (* 1 byte*)
	
END_STRUCT
END_TYPE

// ---- DUTs/Magnemotion/ST_B8Res.TcDUT
(* B8 = Reset *)
TYPE ST_B8Res :
STRUCT
	PathID			:UINT;		(* 2 bytes*)
	CRC1			:BYTE;	    (* 1 byte*)
	CRC2			:BYTE;	    (* 1 byte*)			
END_STRUCT
END_TYPE

// ---- DUTs/Magnemotion/ST_MM_Header.TcDUT
TYPE ST_MM_Header :
STRUCT
	StartBytes	:WORD :=16#ABBA;
	MsgLength	:BYTE :=0;
END_STRUCT
END_TYPE

// ---- DUTs/Magnemotion/ST_MM_ResDataNamed.TcDUT
TYPE ST_MM_ResDataNamed :
STRUCT
	//ResHeader   :ST_MM_ResHeader;
	ResCmdData	:U_MM_ResCmdDataDetail;	
END_STRUCT
END_TYPE

// ---- DUTs/Magnemotion/ST_MM_ResHeader.TcDUT
TYPE ST_MM_ResHeader :
STRUCT
	ResHeader   :BYTE;	
END_STRUCT
END_TYPE

// ---- DUTs/Magnemotion/ST_MM_RxFrame.TcDUT
TYPE ST_MM_RxFrame :
STRUCT
	//head 	:ST_MM_Header;	
	StartBytes	:WORD 	:=16#ABBA;
	MsgLength	:BYTE 	:=0;
	ResHeader   :BYTE	:=0;	
	Resdata :U_MM_ResData;
END_STRUCT
END_TYPE

// ---- DUTs/Magnemotion/ST_MM_TxFrame.TcDUT
TYPE ST_MM_TxFrame :
STRUCT
	//head 	:ST_MM_Header;
    StartBytes	:WORD :=16#ABBA;
	MsgLength	:BYTE :=0;
	DataArray	:ARRAY[0..31] OF BYTE;
	//Cmd_Header	:BYTE ;	
	//Cmddata :U_MM_CmdData;
		
END_STRUCT
END_TYPE

// ---- DUTs/Magnemotion/ST_ResD0.TcDUT
TYPE ST_ResD0 :
STRUCT
	Cmd				:BYTE;
	CmdStatus		:BYTE;
	Cmd_Data_Detail : U_MM_ResD0CmdDataDetail;
END_STRUCT
END_TYPE

// ---- DUTs/Magnemotion/ST_ResD1.TcDUT
TYPE ST_ResD1 :
STRUCT
	HLC_State		:BYTE;
	EIP_Comm_State	:BYTE;		
	CRC1			:BYTE;	    (* 1 byte*)
	CRC2			:BYTE;	    (* 1 byte*)		
END_STRUCT
END_TYPE

// ---- DUTs/Magnemotion/ST_ResD2.TcDUT
TYPE ST_ResD2 :
STRUCT
	Node_Cntl_ID		:UINT;
	Node_Cntl_Present	:BYTE;
	Node_Cntl_State		:BYTE;
	CRC1				:BYTE;	    (* 1 byte*)
	CRC2				:BYTE;	    (* 1 byte*)
END_STRUCT
END_TYPE

// ---- DUTs/Magnemotion/ST_ResD3.TcDUT
TYPE ST_ResD3 :
STRUCT
	Node_Cntl_ID		:UINT;
	Node_Cntl_Present	:BYTE;	
	Node_Type			:BYTE;
	VehicleID			:UINT;
	ReqPos				:BYTE;
	ReportPos			:BYTE;
	Flags				:BYTE;
	CRC1				:BYTE;	    (* 1 byte*)
	CRC2				:BYTE;	    (* 1 byte*)
END_STRUCT
END_TYPE

// ---- DUTs/Magnemotion/ST_ResD4.TcDUT
TYPE ST_ResD4 :
STRUCT
	PathID						:UINT;
	PathPresent					:BYTE;
	NumbVehicles				:BYTE;
	PathState					:BYTE;
	PathMoveStatus				:BYTE;
	UpStreamCommLinkStatus		:BYTE;
	DownStreamCommLinkStatus	:BYTE;
	CRC1						:BYTE;	    (* 1 byte*)
	CRC2						:BYTE;	    (* 1 byte*)
END_STRUCT
END_TYPE

// ---- DUTs/Magnemotion/ST_ResD5.TcDUT
TYPE ST_ResD5 :
STRUCT
	VehicleID		:UINT;
	VehiclePresent	:BYTE;
	PathID			:UINT;
	DestPathID		:UINT;
	VehiclePos		:REAL;
	VehicleSpeed	:REAL;
	VehicleCmdType	:BYTE;
	VehicleFlags	:BYTE;
	VehicleCmdPos	:REAL; (* We are not coding the vehicle station which would have overlapped with these bytes*)
	CRC1			:BYTE;	    (* 1 byte*)
	CRC2			:BYTE;	    (* 1 byte*)
END_STRUCT
END_TYPE

// ---- DUTs/Magnemotion/ST_ResD7.TcDUT
TYPE ST_ResD7 :
STRUCT
	PathID			:UINT;
	PathPresent		:BYTE;
	MotorIndex		:BYTE;
	MotorPresent	:BYTE;
	MotorType		:BYTE;
	MotorFaultData	:ARRAY[0..14] OF BYTE;
	CRC1			:BYTE;	    (* 1 byte*)
	CRC2			:BYTE;	    (* 1 byte*)
END_STRUCT
END_TYPE

// ---- DUTs/Magnemotion/ST_VehicleStatus.TcDUT
TYPE ST_VehicleStatus :
STRUCT
	VehicleID			:	UINT; // 2 bytes
	VehiclePresent		:	BYTE; // 1 byte 
	PathID				:	UINT; // 2 bytes 
	DestinationPathID	:	UINT; // 2 bytes
	VehiclePos			: 	REAL; // 4 bytes
	Velocity			: 	REAL; // 4 bytes 
	VehicleCmdType		: 	BYTE; // 1 byte
	VehicleFlags		: 	BYTE; // 1 byte
	VehicleCmdPos		: 	REAL; // 4 bytes
	junk				:   BYTE; // 1 byte
END_STRUCT
END_TYPE

// ---- DUTs/Magnemotion/ST_VehicleStatusHMI.TcDUT
TYPE ST_VehicleStatusHMI :
STRUCT  
  VehicleStatusBytes  : ARRAY[0..20] OF BYTE;
    (*
	VehicleID			:	UINT; // 2 bytes
	VehiclePresent		:	BYTE; // 1 byte 
	PathID				:	UINT; // 2 bytes 
	DestinationPathID	:	UINT; // 2 bytes
	VehiclePos			: 	REAL; // 4 bytes
	Velocity			: 	REAL; // 4 bytes 
	VehicleCmdType		: 	BYTE; // 1 byte
	VehicleFlags		: 	BYTE; // 1 byte
	VehicleCmdPos		: 	REAL; // 4 bytes
	*)
END_STRUCT
END_TYPE

// ---- DUTs/Magnemotion/U_MM_CmdData.TcDUT
TYPE U_MM_CmdData :
UNION
	
	B1Cmd		:ST_B1Cmd;     
	B2Cmd		:ST_B2Cmd;
	B3Cmd		:ST_B3Cmd;
	B4Cmd		:ST_B4Cmd;
	B5Cmd		:ST_B5Cmd;
	B8Cmd		:ST_B8Cmd;	
END_UNION
END_TYPE

// ---- DUTs/Magnemotion/U_MM_ResCmdDataDetail.TcDUT
TYPE U_MM_ResCmdDataDetail :
UNION	
	D0Res		:ST_ResD0;
    D1Res		:ST_ResD1;     
	D2Res		:ST_ResD2;
	D3Res		:ST_ResD3;
	D4Res		:ST_ResD4;
	D5Res		:ST_ResD5;
	D7Res		:ST_ResD7;	
END_UNION
END_TYPE

// ---- DUTs/Magnemotion/U_MM_ResD0CmdDataDetail.TcDUT
TYPE U_MM_ResD0CmdDataDetail :
UNION	
	B1Res		:ST_B1Res;     
	B2Res		:ST_B2Res;
	B3Res		:ST_B3Res;
	B4Res		:ST_B4Res;	
	B8Res		:ST_B8Res;	
END_UNION
END_TYPE

// ---- DUTs/Magnemotion/U_MM_ResData.TcDUT
TYPE U_MM_ResData :
UNION
	DataArray	:ARRAY[0..31] OF BYTE;
	//Response 	:ST_MM_ResDataNamed;
	ResCmdData	:U_MM_ResCmdDataDetail;		
END_UNION
END_TYPE

// ---- DUTs/PartsDataDUTs/ePartStatus.TcDUT
{attribute 'qualified_only'}
{attribute 'strict'}
TYPE ePartStatus :
(
	eEmpty :=0, // grey
    eLoaded,    // blue 
	eVisionPass, // green 
	ePistonInserted, // green
	eCapInserted, //green 
	eGoodPremium, //green 
	eGoodRegular, // lime green
	eReject, //red
    eJam //vehicle jam
	
);
END_TYPE

// ---- DUTs/PartsDataDUTs/PartDataType.TcDUT
TYPE PartDataType:
STRUCT
	OverallStatus: ePartStatus;	// This will keep getting updated as the part travels and this is used by the machine
	VisionData: VisionInspectDataType; // Data to be recorded to database
	PistonStroke : REAL; // Piston stroke for database
	CapTorque    : REAL; // Cap torque for database     
	Premium 	 : BOOL; // Is Premium
	Good		 : BOOL; // If not premium, but good
	VisionPass	 : BOOL; // If not premium and not good
	PistonPass	 : BOOL; // Piston Pass = 1, 0 if not. Piston Sta be may be disabled, and this value will be 0 even for disabled
	CapPass		 : BOOL; // Cap Pass =1, 0 if failed or station is disabled
	GoodUnload   : BOOL; // Pass =1 if unloaded succesfully, or 0 if not successful or disabled
	PartNumber   : STRING; // Comes from the Part number when started a new Lot
	LotNumber 	 : STRING; // Comes from Lot start 
	LoadTime	 : STRING; //Timestamp when loaded 
	VisionInspectTime : STRING; //Timestamp when vision inspected
	PistonInsertTime : STRING; //Timestamp when piston inserted
	CapInsertTime : STRING; // Timestamp when cap inserted
	RejectUnloadTime : STRING; //Timestamp when reject part is unloaded
    UnloadTime   : STRING; // Timestamp when unloaded ( this for good unload station)
	CavityNumber : INT; // Based on Yushin Position
	BarrelSize	 : eBarrelType; 
	BurnOffTemp  : REAL;
	
END_STRUCT
END_TYPE

// ---- DUTs/PartsDataDUTs/VisionInspectDataType.TcDUT
TYPE VisionInspectDataType :
STRUCT
	Cam1Judgement : BOOL;
	Cam2Judgement : BOOL;
	Cam3Judgement : BOOL;
	Cam4Judgement : BOOL;
	//Short Shot
    MaxIndividualStainArea		   : REAL;
	MinIndividualStainArea	 		 : REAL;
	ModifiedStainArea	 : REAL;
	ModifiedMaxStain     : REAL;
	XPosCam1			 : REAL;
	YPosCam1			 : REAL;
	//Stain
	UpperFlawAreaCam2	  :DINT;
	LowerFlawAreaCam2	 : DINT;
	UpperFlawCountCam2	 : DINT;
	LowerFlawCountCam2	 : DINT;
	XPosAdjustCam2		 : REAL;
	UpperFlawAreaCam3	 : DINT;
	LowerFlawAreaCam3	 : DINT;
	UpperFlawCountCam3	 : DINT;
	LowerFlawCountCam3	 : DINT;
	XPosAdjustCam3		 : REAL;
	UpperFlawAreaCam4	 : DINT;
	LowerFlawAreaCam4	 : DINT;
	UpperFlawCountCam4	 : DINT;
	LowerFlawCountCam4	 : DINT;
	XPosAdjustCam4		 : REAL;
	
END_STRUCT
END_TYPE

// ---- GVLs/CONFIG.TcGVL
{attribute 'qualified_only'}
VAR_GLOBAL PERSISTENT 
	BU_BLOWER_OFF_TIMER : REAL;
    BU_BLOWER_SETPOINT	 : REAL;
 //   BU_HEATER_SETPOINT	 : REAL;
	BU_P_GAIN :REAL;
	BU_I_GAIN :REAL;
	BU_D_GAIN :REAL;
	PremiumCount1 : UINT := 0;
	PremiumCount2 : UINT := 0;
	GoodCount1 : UINT := 0;
	GoodCount2 : UINT := 0;
END_VAR

VAR_GLOBAL
	CAP_INSTALL_RETRIES : BYTE := 2;
    CAP_PICKUP_RETRIES : BYTE := 3;	
END_VAR

VAR_GLOBAL CONSTANT
	MAX_CAVITY : BYTE := 16;
	MAX_CSV_ROWS : DWORD := 50000; // more than a three shifts worth of data
	MAX_CSV_COLUMNS : BYTE := 50;
	MAX_CSV_FIELD_LENGTH : BYTE := 100;
END_VAR

VAR_GLOBAL CONSTANT
	HMI_STATIONS_NUMB : BYTE :=22;
END_VAR

// ---- GVLs/GVL_IO.TcGVL
{attribute 'qualified_only'}
VAR_GLOBAL
	
(* INPUTS *)


    //Bagger Inputs 
    BG_XBaggerBusy      		AT %I* : BOOL;  //Bagger Ready Input --- > need to remove this 
	BG_XBagsLow         		AT %I* : BOOL;  //Bags Low
	BG_XBaggerOKNoFault 		AT %I* : BOOL;  //Bagger Not Faulted
	BG_XBaggerReadyForFiller 	AT %I* : BOOL;  //Bagger Ready For Filler
	BG_XBaggerWaitingForLabel 	AT %I* : BOOL;  //Bagger Waiting For Label
	
	BG_XChute1Open AT %I* : BOOL;
	BG_XChute2Open AT %I* : BOOL;
	BG_XChute3Open AT %I* : BOOL;
	BG_XChute4Open AT %I* : BOOL;
	BG_XChute1Closed AT %I* : BOOL;
	BG_XChute2Closed AT %I* : BOOL;
	BG_XChute3Closed AT %I* : BOOL;
	BG_XChute4Closed AT %I* : BOOL;
	
	
	
 	// Burn Off Inputs
	BU_XAlarm AT %I* : BOOL; //Burn Off Alarm
	BU_Temperature AT %I* :INT; // Burn off Thermocouple
	
	//Cap Insert Inputs
	CP_XPalletHoldDownHome AT %I* : BOOL; // Cap Pallet Hold Down Home
	CP_XPalletHoldDownExtended AT %I* : BOOL; // Cap Pallet HoldDown Extended
	CP_XCapSlideRetracted AT %I* : BOOL; // Cap Slide Retracted Sensor
	CP_XCapSlideExtended AT %I* : BOOL; // CapSlide Extended Sensor
	
	//Good Unload Inputs
	UL_XGrippersOpened AT %I* : BOOL; //Good Unload Grippers Opened
	UL_XGrippersClosed AT %I* : BOOL; //Good Unload Grippers Closed
//	UL_XPalletReleaseHome AT %I* : BOOL; // Pallet Release Retracted 
//	UL_XPalletReleaseExtended AT %I* : BOOL; // Pallet Release Extended
	UL_XRotatorCWBarrelLeftBin AT %I* : BOOL; // Rotator to Left Bin
	UL_XRotatorCWBarrelRightBin AT %I* : BOOL; //Rotator to Right Bin 
	UL_XRotatorCenter AT %I* : BOOL; // Rotator Center Position
	
	UL_XBarrelPresent AT %I* : BOOL; //UL Barrel Present
	UL_XPalletHoldDownRetracted_Engaged AT %I* : BOOL; // Unload Pallet Hold Down Home
	UL_XPalletHoldDownExtended_Home AT %I* : BOOL; // Unload Pallet HoldDown Extended
	
	UL_1_XBarrelPresent AT %I* : BOOL; //UL Barrel Present
	UL_1_XPalletHoldDownRetracted_Engaged AT %I* : BOOL; // Unload Pallet Hold Down Home
	UL_1_XPalletHoldDownExtended_Home AT %I* : BOOL; // Unload Pallet HoldDown Extended
	UL_2_XBarrelPresent AT %I* : BOOL; //UL Barrel Present
	UL_2_XPalletHoldDownRetracted_Engaged AT %I* : BOOL; // Unload Pallet Hold Down Home
	UL_2_XPalletHoldDownExtended_Home AT %I* : BOOL; // Unload Pallet HoldDown Extended
	UL_3_XBarrelPresent AT %I* : BOOL; //UL Barrel Present
	UL_3_XPalletHoldDownRetracted_Engaged AT %I* : BOOL; // Unload Pallet Hold Down Home
	UL_3_XPalletHoldDownExtended_Home AT %I* : BOOL; // Unload Pallet HoldDown Extended
	UL_4_XBarrelPresent AT %I* : BOOL; //UL Barrel Present
	UL_4_XPalletHoldDownRetracted_Engaged AT %I* : BOOL; // Unload Pallet Hold Down Home
	UL_4_XPalletHoldDownExtended_Home AT %I* : BOOL; // Unload Pallet HoldDown Extended
	
	UL_XPP_DriveEnabled 	: 	BOOL; // Drive Enabled or not
	UL_XPP_StopActive		:	BOOL; // Is Stop Active
	UL_XPP_ReferenceOK		:	BOOL; // Is reference (home) OK? Without this, sequence will not execute
	UL_XPP_ReadyToStart		:	BOOL; // Is Drive Ready to Start
	UL_XPP_InPos			: 	BOOL; // Last Move in Pos
	UL_XPP_Alarm			: 	BOOL; // Alarm in Drive 
	UL_XPP_A1OUT			:	BOOL; // Out A1 from Sequence
	UL_XPP_A2OUT			:	BOOL; // Out A2 from Sequence
	UL_XPP_A3OUT			:	BOOL; // Out A3 from Sequence
	UL_XPP_ReqLubeON		:	BOOL; // Connect this to the Lube Valve
	UL_XPP_LubeLevel		:	BOOL; // PP is mirroring lube level 
	
	
	UL_XPP_Byte4 AT %I*		: BYTE;
	UL_XPP_Byte5 AT %I*		: BYTE;
	// Inonizer Inputs
	IZ_XIonAlarm AT %I* : BOOL; //Ionizer Alarm
	IZ_XConditionAlarm AT %I* : BOOL; //Condition Alarm
	IZ_XAlarm AT %I* : BOOL; //Alarm
	
	// Load Position Inputs
	LD_XPalletHoldRetractEngage AT %I* : BOOL;  //Load Pallet HoldDown Home
	LD_XPalletHoldDownExtendHome AT %I* : BOOL;  // Load Pallet HoldDown Extended
	LD_XPalletReleaseHome AT %I* : BOOL;  //Load Pallet Release Retracted
	LD_XPalletReleaseExtended AT %I* : BOOL;  //Load PalletRelease Extended
	LD_XPalletCloseRetracted_1_2 AT %I* : BOOL; //Load Pallet Release Retract
	LD_XPalletCloseExtended_1_2 AT %I*: BOOL; //Load PalletRelease Extended
	LD_XPalletCloseRetracted_3_4 AT %I* : BOOL; //Load Pallet Release Retract
	LD_XPalletCloseExtended_3_4 AT %I*: BOOL; //Load PalletRelease Extended
	
	
	
	// Main Control System 
	
	MC_XAirPressureOK AT %I* : BOOL; //Air Pressure OK
	MC_XStartPB AT %I* : BOOL;  // Start PB
	MC_XStopPB AT %I* : BOOL;  //Stop PB	
	//MC_NotEStopped AT %I* : BOOL; // Output from switched 24V. D.C. (TRUE := NO E-STOP, FALSE := E-STOPPED)
	MC_NotEStopped AT %I* : BOOL; // Output from switched 24V. D.C. (TRUE := NO E-STOP, FALSE := E-STOPPED)
	MachineEStopped : BOOL;
	
    //Piston Insert 
	
	PI_XPalletHoldDownHome AT %I* : BOOL;  // Piston Pallet Hold Down Retracted 
	PI_XPalletHoldDownExtended AT %I* : BOOL; //Piston Pallet Hold Down Extended
	PI_XPistonPresentEscapement AT %I* : BOOL;  //Part Present in Escapement
	PI_XEscapementAtInsertLoc AT %I* : BOOL;  //Escapement at Insert Location
	PI_XEscapementAtBowl AT %I* : BOOL;  //Escapement is at Bowl Location
	PI_XToolAt55_10_Barrel AT %I* : BOOL;  //Tool is at 55 cc Location
	PI_XToolAt3_30_Barrel AT %I* : BOOL;  //Tool is at 3 and 30 cc Location
	PI_XBarrelHoldDownHome AT %I* : BOOL;  //Barrel Hold Down at Home Location
	PI_XBarrelHoldDownExtended AT %I* : BOOL;  //Barrel Hold Down at Part
	
	PI_XMtrOUT0 : BOOL; // Out 0 From SMC LEY JXC91 Ethernet IP Controller
	PI_XMtrOUT1 : BOOL; // Out 1 From SMC LEY JXC91 Ethernet IP Controller
	PI_XMtrOUT2 : BOOL; // Out 2 From SMC LEY JXC91 Ethernet IP Controller
	PI_XMtrOUT3 : BOOL; // Out 3 From SMC LEY JXC91 Ethernet IP Controller
	PI_XMtrOUT4 : BOOL; // Out 4 From SMC LEY JXC91 Ethernet IP Controller
	PI_XMtrOUT5 : BOOL; // Out 5 From SMC LEY JXC91 Ethernet IP Controller
	PI_XMtrBusy : BOOL; // Piston Insert Stepper Busy
	PI_XMtrServoEnabled : BOOL; // Pistion Stepper Enabled
	PI_XMtrServoHomed : BOOL; //Piston Stepper Homed
	PI_XMtrMoveCompl: BOOL; //Piston Stepper Move complete
	PI_XMtrEStopped : BOOL; //Piston Motor E-Stopped
	PI_XMtrAlarm : BOOL; // Piston Motor Alarm
	PI_XMtrReady : BOOL; // Pistom Motor Ready Bit from SMC LEY JXCP1 EIP
	
	PI_XMtrCurrPos : REAL;
	
	// Reject Unload 
	
	RJ_XRejectCylinderHome AT %I* : BOOL;  //Reject Cyclinder at home location
	RJ_XRejectCylinderExtended AT %I* : BOOL;  //Reject Cylinder extended location
//	RJ_XPalletReleaseHome AT %I* : BOOL;  // Reject Pallet Release Home
//	RJ_XPalletReleaseExtended AT %I* : BOOL;  //Reject Pallet Release Extended 
	RJ_XPartPresent AT %I* : BOOL; //Reject Part Present Sensor PhotoEye
	RJ_XPalletHoldDownExtended_Home AT %I* : BOOL; // Reject Pallet Horizontal Locater Extended
	RJ_XPalletHoldDownRetracted_Engaged AT %I* : BOOL; // Reject Pallet Horizontal Locater Retracted
	
	//Yushin Robot Interface Inputs
	YU_XPrepareToLoad AT %I* : BOOL;  //Prepare Track to Load Parts
	YU_XToolUp AT %I* : BOOL;  //Tool is up, clear to move
	YU_XToolDown AT %I* : BOOL;  //Tool is down, parts are transferred
	YU_XLocBit0 AT %I* : BOOL;  //Location Bit 0 
	YU_XLocBit1 AT %I* : BOOL; //Location Bit 1 
	
	
	//Vision
	VS_XToolingLocationUpper AT %I* : BOOL;  //Vision Tooling sensor location at upper height
	VS_XToolingLocationLower AT %I* : BOOL; // Vision Tooling sensor location at lower height 
	VS_XCmdCmpl : BOOL; // Turns ON when command processing is complete
	VS_XCmdErr  : BOOL; // Turns OFF when command processing is successful and turns ON when it fails
	VS_XCmdReady : BOOL; // Turns ON when command processes can be received
	VS_XCmdResult : BYTE;
	VS_XCmdData1 : BYTE;
	VS_XCmdData2 : BYTE;
	VS_XResultReady : BOOL; // Turns ON when data processing is complete
	VS_XResultOR : BOOL; // Used to output the OR result for the judged value of the tools specified in the output settings
	VS_XReady1 : BOOL; // Signals the Trigger 1 is acceptable
	VS_XReady2 : BOOL; // Signals the Trigger 2 is acceptable
	VS_XReady3 : BOOL; // Signals the Trigger 3 is acceptable
	VS_XReady4 : BOOL; // Signals the Trigger 4 is acceptable
	VS_XAck1 : BOOL; // Turns ON when Trigger 1 is accepted. Turns OFF when Trigger 1 is set to OFF
	VS_XAck2 : BOOL; // Turns ON when Trigger 1 is accepted. Turns OFF when Trigger 1 is set to OFF
	VS_xAck3 : BOOL; // Turns ON when Trigger 1 is accepted. Turns OFF when Trigger 1 is set to OFF
	VS_XAck4 : BOOL; // Turns ON when Trigger 1 is accepted. Turns OFF when Trigger 1 is set to OFF
	VS_XBusy : BOOL; // When Command Processing or Image Processing
	VS_XError : BOOL; // Any system errors
    VS_XRun  : BOOL; // When in Run Mode
	VS_XAllCamJudgeVal: BOOL; //All Camera Judgement Values
	VS_XCam1JudgeVal: BOOL; // Camera 1 Judgement Value...set this up in the Judgement top level selection in the output config at the Keyence controller
	VS_XCam2JudgeVal: BOOL; // Camera 2 Judgement Value...set this up in the Judgement top level selection in the output config at the Keyence controller
	VS_XCam3JudgeVal: BOOL; // Camera 3 Judgement Value...set this up in the Judgement top level selection in the output config at the Keyence controller
	VS_XCam4JudgeVal: BOOL; // Camera 4 Judgement Value .. set this up in the Judgement top level selection in the output config at the Keyence controller
	VS_XPartEmpty : BOOL;  // Will be 1 when empty and 0 wehn present 0:4
	VS_XPartPresentBeforeVision  AT %I* : BOOL; // New Part Present Sensor before Vision Station
	
	//Short Shot
    VS_XMaxIndividualStainArea  : REAL;
	VS_XMinIndividualStainArea	: REAL;
	VS_XModifiedStainArea		: REAL;
	VS_XModifiedMaxStain        : REAL;
	VS_XXPosCam1				: REAL;
	VS_XYPosCam1		 		: REAL;
	//Stain
	VS_XUpperFlawAreaCam2	 	: DINT;
	VS_XLowerFlawAreaCam2	 	: DINT;
	VS_XUpperFlawCountCam2	 	: DINT;
	VS_XLowerFlawCountCam2	 	: DINT;
	VS_XXPosAdjustCam2		 	: REAL;
	VS_XUpperFlawAreaCam3	 	: DINT;
	VS_XLowerFlawAreaCam3	 	: DINT;
	VS_XUpperFlawCountCam3	 	: DINT;
	VS_XLowerFlawCountCam3	 	: DINT;
	VS_XXPosAdjustCam3		 	: REAL;
	VS_XUpperFlawAreaCam4	 	: DINT;
	VS_XLowerFlawAreaCam4	 	: DINT;
	VS_XUpperFlawCountCam4	 	: DINT;
	VS_XLowerFlawCountCam4	 	: DINT;
	VS_XXPosAdjustCam4		 	: REAL;
	
	
	VS_XByte0 AT %I* : BYTE; // Vision Byte 0
	VS_XByte1 AT %I* : BYTE; // Vision Byte 1
	VS_XByte2 AT %I* : BYTE; // Vision Byte 2
	VS_XByte3 AT %I* : BYTE; // Vision Byte 3
	VS_XByte4 AT %I* : BYTE; // Vision Byte 4

	VS_XByte20 AT %I* : BYTE; //Vision Byte 20
	VS_XByte24 AT %I* : BYTE; //Vision Byte 24
	VS_XByte28 AT %I* : BYTE; //Vision Byte 28
	
	VS_XByte48 AT %I* : BYTE; //Vision Byte 48
	VS_XByte49 AT %I* : BYTE; //Vision Byte 48
	VS_XByte50 AT %I* : BYTE; //Vision Byte 48
	VS_XByte51 AT %I* : BYTE; //Vision Byte 48
	
	VS_XByte52 AT %I* : BYTE; //Vision Byte 52
	VS_XByte53 AT %I* : BYTE; //Vision Byte 53
	VS_XByte54 AT %I* : BYTE; //Vision Byte 54
	VS_XByte55 AT %I* : BYTE; //Vision Byte 55
	
	VS_XByte56 AT %I* : BYTE; //Vision Byte 56
	VS_XByte57 AT %I* : BYTE; //Vision Byte 57
	VS_XByte58 AT %I* : BYTE; //Vision Byte 58
	VS_XByte59 AT %I* : BYTE; //Vision Byte 59
	
	VS_XByte60 AT %I* : BYTE; //Vision Byte 60
	VS_XByte61 AT %I* : BYTE; //Vision Byte 61
	VS_XByte62 AT %I* : BYTE; //Vision Byte 62
	VS_XByte63 AT %I* : BYTE; //Vision Byte 63
	
	VS_XByte64 AT %I* : BYTE; //Vision Byte 64
	VS_XByte65 AT %I* : BYTE; //Vision Byte 65
	VS_XByte66 AT %I* : BYTE; //Vision Byte 66
	VS_XByte67 AT %I* : BYTE; //Vision Byte 67
	
	VS_XByte68 AT %I* : BYTE; //Vision Byte 68
	VS_XByte69 AT %I* : BYTE; //Vision Byte 69
	VS_XByte70 AT %I* : BYTE; //Vision Byte 70
	VS_XByte71 AT %I* : BYTE; //Vision Byte 71
	                                          
	VS_XByte72 AT %I* : BYTE; //Vision Byte 72
	VS_XByte73 AT %I* : BYTE; //Vision Byte 73
	VS_XByte74 AT %I* : BYTE; //Vision Byte 74
	VS_XByte75 AT %I* : BYTE; //Vision Byte 75
	                                          
	VS_XByte76 AT %I* : BYTE; //Vision Byte 76
	VS_XByte77 AT %I* : BYTE; //Vision Byte 77
	VS_XByte78 AT %I* : BYTE; //Vision Byte 78
	VS_XByte79 AT %I* : BYTE; //Vision Byte 79
	                                          
	VS_XByte80 AT %I* : BYTE; //Vision Byte 80
	VS_XByte81 AT %I* : BYTE; //Vision Byte 81
	VS_XByte82 AT %I* : BYTE; //Vision Byte 82
	VS_XByte83 AT %I* : BYTE; //Vision Byte 83
	
	VS_XByte88 AT %I* : BYTE; //Vision Byte 88 
	VS_XByte89 AT %I* : BYTE; //Vision Byte 89 
	VS_XByte90 AT %I* : BYTE; //Vision Byte 90 
	VS_XByte91 AT %I* : BYTE; //Vision Byte 91 
	                                           
	VS_XByte92 AT %I* : BYTE; //Vision Byte 92 
	VS_XByte93 AT %I* : BYTE; //Vision Byte 93 
	VS_XByte94 AT %I* : BYTE; //Vision Byte 94 
	VS_XByte95 AT %I* : BYTE; //Vision Byte 95 
	                                           
	VS_XByte96 AT %I* : BYTE; //Vision Byte 96 
	VS_XByte97 AT %I* : BYTE; //Vision Byte 97 
	VS_XByte98 AT %I* : BYTE; //Vision Byte 98 
	VS_XByte99 AT %I* : BYTE; //Vision Byte 99 
	                                           
	VS_XByte100 AT %I* : BYTE; //Vision Byte 100
	VS_XByte101 AT %I* : BYTE; //Vision Byte 101
	VS_XByte102 AT %I* : BYTE; //Vision Byte 102
	VS_XByte103 AT %I* : BYTE; //Vision Byte 103

	VS_XByte108 AT %I* : BYTE; //Vision Byte 108 
	VS_XByte109 AT %I* : BYTE; //Vision Byte 109 
	VS_XByte110 AT %I* : BYTE; //Vision Byte 110 
	VS_XByte111 AT %I* : BYTE; //Vision Byte 111 
	                                             
	VS_XByte112 AT %I* : BYTE; //Vision Byte 112 
	VS_XByte113 AT %I* : BYTE; //Vision Byte 113 
	VS_XByte114 AT %I* : BYTE; //Vision Byte 114 
	VS_XByte115 AT %I* : BYTE; //Vision Byte 115 
	                                             
	VS_XByte116 AT %I* : BYTE; //Vision Byte 116 
	VS_XByte117 AT %I* : BYTE; //Vision Byte 117 
	VS_XByte118 AT %I* : BYTE; //Vision Byte 118 
	VS_XByte119 AT %I* : BYTE; //Vision Byte 119 
	                                             
	VS_XByte120 AT %I* : BYTE; //Vision Byte 120 
	VS_XByte121 AT %I* : BYTE; //Vision Byte 121 
	VS_XByte122 AT %I* : BYTE; //Vision Byte 122 
	VS_XByte123 AT %I* : BYTE; //Vision Byte 123                                         
	
	
	
      
	
(* OUTPUTS *)

	
	//Bagger Outputs
  	BG_YFillerTrigger AT %Q* : BOOL;   //Feeder Ready Ouput, also called Filler Trigger in Sharp Docs
	BG_YOpenChute1 AT %Q* : BOOL;
	BG_YOpenChute2 AT %Q* : BOOL;
	BG_YOpenChute3 AT %Q* : BOOL;
	BG_YOpenChute4 AT %Q* : BOOL;
	BG_YCloseChute1 AT %Q* : BOOL;
	BG_YCloseChute2 AT %Q* : BOOL;
	BG_YCloseChute3 AT %Q* : BOOL;
	BG_YCloseChute4 AT %Q* : BOOL;
	
	//Burn Off Outputs
	BU_HeatCntl AT %Q* :INT; // Burn off Heater
	BU_BlowCntl AT %Q* :INT; // Burn off Heater
	
	//Cap Insert Outputs
	(*
	CP_YSMAC0 AT %Q* : BOOL; //SMAC Output 1
	CP_YSMAC1 AT %Q* : BOOL; // SMAC Output 2
	CP_YSMAC2 AT %Q* : BOOL; // SMAC Output 2
	CP_YSMAC3 AT %Q* : BOOL; // SMAC Output 2	
	CP_YEscapeWallCylinderExtend : BOOL; //Cap Escapement Wall Extended
	CP_YEscapeWallCylinderRetract : BOOL; // Cap Escapement Wall Retracted
	CP_YEscapementToPick : BOOL; //Cap Escapement to Pickup location
	CP_YEscapementToBowl : BOOL; //Cap Escapement to Bowl Location

	CP_YToolVacuumON AT %Q*: BOOL; //Vacuum ON
	CP_YToolVacuumOFF AT %Q*: BOOL; //Vacuum OFF
	CP_YBarellCenterPinExtend : BOOL; // Cap Barrel Center Pin Extend/Raise to center the barrel
	CP_YBarellCenterPinRetract : BOOL; // Cap Barrel Center Pin Lower to center the barrel
	*)
	CP_YCapSlideExtend : BOOL;  //Cap Slide Extend and Torque
    CP_YCapSlideRetract : BOOL; //Cap Slide Retract 
	CP_YPalletHoldDownExtend: BOOL; //Cap Hold Down pallet
	CP_YPalletHoldDownRetract : BOOL; //Cap Retract Pallet Hold down	
	
	//Good Unload Outputs
	
	UL_YGrippersOpen : BOOL; //Good Unload Open Grippers
	UL_YGrippersClose: BOOL; // Good Unload Close Grippers
	UL_YRotatorCCWBarrelRightBin : BOOL; //Rotate Gripper to Right Bin
	UL_YRotatorCWBarrelLeftBin: BOOL;
//	UL_YPalletReleaseExtend: BOOL; 
//	UL_YPalletReleaseRetract : BOOL;
    UL_YPalletHoldDownExtend_Home : BOOL;
    UL_YPalletHoldDownRetract_Engage : BOOL;
	
	UL_1_YPalletHoldDownExtend_Home : BOOL;
    UL_1_YPalletHoldDownRetract_Engage : BOOL;
	UL_1_YRejectPushExtend  : BOOL; 
	UL_1_YRejectPushRetract : BOOL; 
	
	UL_2_YPalletHoldDownExtend_Home : BOOL;
    UL_2_YPalletHoldDownRetract_Engage : BOOL;
	UL_2_YRejectPushExtend  : BOOL; 
	UL_2_YRejectPushRetract : BOOL; 
	
	UL_3_YPalletHoldDownExtend_Home : BOOL;
    UL_3_YPalletHoldDownRetract_Engage : BOOL;
	UL_3_YRejectPushExtend  : BOOL; 
	UL_3_YRejectPushRetract : BOOL; 
	
	UL_4_YPalletHoldDownExtend_Home : BOOL;
    UL_4_YPalletHoldDownRetract_Engage : BOOL;
	UL_4_YRejectPushExtend  : BOOL; 
	UL_4_YRejectPushRetract : BOOL; 
	
	
	UL_YPP_Enable		:	BOOL;
	UL_YPP_Stop			:	BOOL;
	UL_YPP_ResetAlarm	:	BOOL;
	UL_YPP_StartHoming	:	BOOL;
	UL_YPP_StartSeq		:	BOOL;
	UL_YPP_BitA			:	BOOL;
	UL_YPP_BitB			:	BOOL;
	UL_YPP_BitC			:	BOOL;
	
	UL_YPP_Byte4   AT %Q* : BYTE;
					
	
	
	
	//Ionizer Outputs
	
	IZ_YInterrupt AT %Q* : BOOL; // Interrupt Ionizer Output
	//IZ_YIonizerAirON : BOOL;
	//IZ_YIonizerAirOFF : BOOL;
	
	//Load Position Outputs
	LD_YPalletHoldDownExtendHome : BOOL; //Load Pallet Hold Down Extend
	LD_YPalletHoldDownRetractEngage : BOOL; //Load Pallet Hold Down Retract
	LD_YPalletReleaseExtend :BOOL; //Load Pallet Center Pin Extend
	LD_YPalletReleaseRetract : BOOL; //Load Pallet Center Pin Retract
	LD_YPalletCloseExtend :BOOL; //Load PalletRelease Extend
	LD_YPalletCloseRetract : BOOL; //Load Pallet Release Retract
	
	//Main Control System
	
	MC_YStackLightYellow AT %Q* : BOOL;  // Yellow Stack Light
	MC_YStackLightRed AT %Q* :  BOOL; //Red Stack Light
	MC_YStackLightGreen AT %Q* : BOOL; //Green Stack Light
	
	// Vision
	
	VS_YBarrelLED : BOOL; //Vison LED for Barrel Advanced Illumination
	VS_YBarrelLED_off AT %Q* : BOOL; //Vison LED for Barrel Advanced Illumination
	VS_YCmdRequest : BOOL; // Provides command execution when signal switches from OFF to ON
	VS_YResultAck : BOOL; // Provides notification of data acquisition when signal swtiches from OFF to ON
	VS_YErrorReset : BOOL; // Clears Error when signal switches from OFF to ON
	VS_YTrigger1 : BOOL; // Trigger Camera 1, note Ready 1 must be ON prior to issuing trigger
	VS_YTrigger2 : BOOL; // Trigger Camera 2, note Ready 2 must be ON prior to issuing trigger
	VS_YTrigger3 : BOOL; // Trigger Camera 3, note Ready 3 must be ON prior to issuing trigger
	VS_YTrigger4 : BOOL; // Trigger Camera 4, note Ready 4 must be ON prior to issuing trigger
	VS_YCmdNumber : BYTE; // This maps into DWORD, but let's limit to BYTE
	VS_YCmdParam1 : BYTE; // This maps into DWORD, but let's limit to BYTE
	VS_YCmdParam2 : BYTE; // This maps into DWORD, but let's limit to BYTE
	VS_YCmdParam3 : BYTE; // This maps into DWORD, but let's limit to BYTE
	
	VS_YByte0 AT %Q* : BYTE;  //contains utility bits including Command Request
	VS_YByte1 AT %Q* : BYTE;  
	VS_YByte2 AT %Q* : BYTE;
    VS_YByte16 AT %Q* : BYTE;  //Command Number
    VS_YByte20 AT %Q* : BYTE;  //Command Parameter 1
    VS_YByte24 AT %Q* : BYTE;  //Param 2

  	
	//Piston Insert 
	
	PI_YPalletHoldDownExtend : BOOL; // Piston Pallet Hold Down
	PI_YPalletHoldDownRetract : BOOL; // Piston Pallet Hold Down Release
	PI_YEscapementToBowl : BOOL; //Piston Move Escapement to Bowl
	PI_YEscapementToWork : BOOL; //Piston Move to Work Location
	PI_YBarrelBackupExtend :BOOL; //Piston Barrel Backup
	PI_YBarrelBackupRetract : BOOL; //Piston Barrel Retract 
	PI_YPistonBowlON: BOOL; // Piston Bowl
	PI_YPistonBowlOFF: BOOL; // Piston Bowl
	
	
	PI_YMtrStepSelectIN0 : BOOL; // INO of SMC JXC91 EtherNet/IP Controller
	PI_YMtrStepSelectIN1 : BOOL; // INO of SMC JXC91 EtherNet/IP Controller
	PI_YMtrStepSelectIN2 : BOOL; // INO of SMC JXC91 EtherNet/IP Controller
	PI_YMtrStepSelectIN3 : BOOL; // INO of SMC JXC91 EtherNet/IP Controller
	PI_YMtrStepSelectIN4 : BOOL; // INO of SMC JXC91 EtherNet/IP Controller
	PI_YMtrStepSelectIN5 : BOOL; // INO of SMC JXC91 EtherNet/IP Controller
	
	PI_YMtrHoldMove : BOOL; // Hold Move of SMC JXC91 EtherNet/IP Controller
	PI_YMtrSetEnable : BOOL; // Enable Stepper Motor
	PI_YMtrDriveStepTrigger : BOOL;  //Trigger Stepper Drive
	PI_YMtrReset : BOOL; // Reset Stepper Motor
	PI_YMtrGoHome : BOOL; // Home Stepper Motor
	PI_YMtrJogPos : BOOL; // Jog Stepper Motor Pos
	PI_YMtrJogNeg : BOOL;  // Jog Stepper Motor Neg
	PI_YMtrSwitchJogInch : BOOL; // Switch Between Inch and Jog Mode

	
	//Prime Mover
	MM_YEnableMagneMotion AT %Q*: BOOL; //New INewnable Magnemotion - this can be tied to safety relay 
	
	//Reject Unload 
	RJ_YRejectPushExtend  : BOOL; 
	RJ_YRejectPushRetract : BOOL; 
//	RJ_YPalletReleaseExtend : BOOL; //Release Pallet extend
//	RJ_YPalletReleaseRetract : BOOL;  //Release Pallet retracted 
	RJ_YPalletHoldDownExtend_Home : BOOL; //Reject Pallet Locater / Holder coming in horizontally Extend/Engage
	RJ_YPalletHoldDownRetract_Engage : BOOL; //Reject Pallet Locater / Holder coming in horizontally Retract/Disengage
	
	//Yushin Robot Interface Outputs
	YU_YOkToLoad AT %Q* : BOOL; //Signal to Yushin OK to Load 
	YU_YAckPartsHeld AT %Q* : BOOL; //Signal that Parts are held
	YU_YIMBADIsOK AT %Q* : BOOL; // Signal that IMABD IS RUNNING
	
	// FieldBus Outputs for instances where Outputs can't be linked directly via I/O linking utility 
	// SMC Does not provide output bits for linking. Note that indexing is 0 based in the software, but Terminal Valve Numbers used in I/O List Document are 1 based indexing 
    SMCEX260_1_Byte0 AT %Q* :BYTE; //
	SMCEX260_1_Byte1 AT %Q* :BYTE; //
	SMCEX260_1_Byte2 AT %Q* :BYTE; //
	SMCEX260_1_Byte3 AT %Q* :BYTE; //
    SMCEX260_2_Byte0 AT %Q* :BYTE; //
	SMCEX260_2_Byte1 AT %Q* :BYTE; //
	SMCEX260_2_Byte2 AT %Q* :BYTE; //
	SMCEX260_2_Byte3 AT %Q* :BYTE; //
	
	SMC_LEY_YUINT0 AT %Q* : UINT;
	//SMC_LEY_YByte0 AT %Q* : BYTE;
	//SMC_LEY_YByte1 AT %Q* : BYTE;
	
	//SMC_LEY_YByte2 AT %Q* : BYTE;
	//SMC_LEY_YByte3 AT %Q* : BYTE;
	
	SMC_LEY_XUINT0 AT %I* : UINT;
	SMC_LEY_XUINT1 AT %I* : UINT;
	SMC_LEY_XCurrMtrPos AT %I* : DINT;
(*	
	SMC_LEY_XByte0 AT %I* : BYTE;
	SMC_LEY_XByte1 AT %I* : BYTE;
	SMC_LEY_XByte2 AT %I* : BYTE;
	SMC_LEY_XByte3 AT %I* : BYTE;
	SMC_LEY_XByte4 AT %I* : BYTE;
	SMC_LEY_XByte5 AT %I* : BYTE;
	SMC_LEY_XByte6 AT %I* : BYTE;
	SMC_LEY_XByte7 AT %I* : BYTE;
*)	
	InputsForHMI : ARRAY[1..128] OF BYTE;
	OutputsForHMI :ARRAY[1..128] OF BYTE;
	OutputsFromHMI: ARRAY[1..128] OF BYTE;
	IOLockedFromHMI : BYTE;
	ResumeMovementFromHMI: BYTE := 0;
	
	RxBufferEL			: ComBuffer;	(* Receive data buffer; used with all receive function blocks *)
	TxBufferEL			: ComBuffer;	(* Transmit data buffer; used with all receive function blocks *)
	
END_VAR

// ---- GVLs/Logging.TcGVL
{attribute 'qualified_only'}
VAR_GLOBAL
	fbEventMsg : EventMsg;
	fbEventMsgParams : EventMsgParams;
	fbCurrTime : FB_LocalSystemTime := (bEnable := TRUE, dwCycle := 1);
END_VAR

VAR_GLOBAL CONSTANT   //Source Constants
	SrcMainPOU 		:UDINT := 1000;
	SrcLoadPOU		:UDINT := 2000;
	SrcVisionPOU	:UDINT := 3000;
	SrcPistonPOU 	:UDINT := 4000;
	SrcCapPOU 		:UDINT := 5000;
	SrcGoodULPOU 	:UDINT := 6000;
	SrcRejectPOU 	:UDINT := 7000;
	SrcBaggerPOU 	:UDINT := 8000;
	SrcMMPOU 		:UDINT := 9000;	
	SrcCyclePOU		:UDINT := 10000;
END_VAR

VAR_GLOBAL CONSTANT   //ID Constants
	


	// Main
	IDMain_InitBegin : UDINT := 1;
	IDMain_InitCmpl  : UDINT := 2;
	IDMain_Tick		 : UDINT := 3;
	IDMain_IOLocked  : UDINT := 4;
	
	//Load
	
	//Vision
	
	//Piston Insert
	// Reserved 1-50 ID for state machine states to be sent 
	ID_PI_Unknown 						: UDINT:=51;
	ID_PI_MtrReset 						: UDINT:=52;
	ID_PI_MtrEnabled					: UDINT:=53;
	ID_PI_MtrCheckEnabled 				: UDINT:=54;
	ID_PI_MtrCheckHome					: UDINT:=55;
	ID_PI_MtrCheckHomePos				: UDINT:=56;
	ID_PI_CheckCylinders 				: UDINT:=57;
	ID_PI_CheckEscapeCylinders	 		: UDINT:=58;
	ID_PI_WaitPiston 					: UDINT:=59;
	ID_PI_WaitVehicle 					: UDINT:=60;
	ID_PI_MtrWaitMoveStart 				: UDINT:=61;
	ID_PI_MtrWaitMoveCmpl 				: UDINT:=62;
	
	// Cap Insert 
	// Reserved 1-50 ID for state machine states to be sent 
	ID_CP_Unknown 						: UDINT:=51;
	ID_CP_MtrReset 						: UDINT:=52;
	ID_CP_MtrEnabled					: UDINT:=53;
	ID_CP_MtrCheckEnabled 				: UDINT:=54;
	ID_CP_MtrCheckHome					: UDINT:=55;
	ID_CP_AllCheckHome					: UDINT:=56;
	ID_CP_CheckCylinders 				: UDINT:=57;
	ID_CP_CheckEscapeCylinders	 		: UDINT:=58;
	ID_CP_WaitCap	 					: UDINT:=59;
	ID_CP_WaitVehicle 					: UDINT:=60;
	ID_CP_MtrWaitCapPickCmpl			: UDINT:=61;
	ID_CP_MtrWaitCapInsertCmpl			: UDINT:=62;
	ID_CP_MtrWaitReturnHomeCmpl			: UDINT:=62;
	
	//Good Unload 
	// Reserved 1-50 ID for state machine states to be sent 
	ID_UL_Unknown 						: UDINT:=51;
	ID_UL_PPReset 						: UDINT:=52;
	ID_UL_PPEnabled						: UDINT:=53;
	ID_UL_PPCheckEnabled 				: UDINT:=54;
	ID_UL_PPCheckHome					: UDINT:=55;	
	ID_UL_PPWaitMoveCmpl				: UDINT:=56;
	ID_UL_PPReady						: UDINT:=57;
	ID_UL_AllCheckHome					: UDINT:=61;
	ID_UL_CheckCylinders 				: UDINT:=62;
	ID_UL_CheckGrippers			 		: UDINT:=63;
	ID_UL_WaitVehicle 					: UDINT:=64;
	
    //Reject Station
		// Reserved 1-50 ID for state machine states to be sent 
	ID_RJ_Unknown 						: UDINT:=51;
	ID_RJ_CheckCylinders 				: UDINT:=52;
	ID_RJ_WaitVehicle 					: UDINT:=53;	
	
	//Load Station
	ID_LD_Unknown 						: UDINT:=51;
	ID_LD_CheckCylinders 				: UDINT:=52;
	ID_LD_WaitVehicle 					: UDINT:=53;	
	
	//Primve Mover
	ID_MM_Unknown 						: UDINT:=51;
	
	//Cycle Control
	ID_CY_Unknown 						: UDINT:=51;
	
	
	//Vision Station
	ID_VS_Unknown						: UDINT:=51;
	ID_VS_CmdProcessNotReady			: UDINT:=52;
	
END_VAR

// ---- GVLs/LotsData.TcGVL
{attribute 'qualified_only'}
VAR_GLOBAL PERSISTENT 
	Lot: LotDataType;
END_VAR

// ---- GVLs/MM_CONST.TcGVL
{attribute 'qualified_only'}
VAR_GLOBAL CONSTANT
	B1_CMD_LEN :BYTE := 26; (* Doesn't Includes 2 Bytes START, 1 byte LEN , includes cmd + 2 Bytes CRC*) //Move Veh to Pos
	B2_CMD_LEN :BYTE := 5; (* Doesn't includes 2 Bytes START, 1 byte LEN, includes cmd + 2 Bytes CRC*) //Startup
	B3_CMD_LEN :BYTE := 8; (* Includes 2 Bytes START, 1 byte LEN + DATA + 2 Bytes CRC*)
	B4_CMD_LEN :BYTE := 8; (* Includes 2 Bytes START, 1 byte LEN + DATA + 2 Bytes CRC*)
	B5_CMD_LEN :BYTE := 7; (* Doesn't includes 2 Bytes START, 1 byte LEN, includes 2 Bytes CRC*) //Status 
	B8_CMD_LEN :BYTE := 5; (* Doesn't includes 2 Bytes START, 1 byte LEN, includes cmd + 2 Bytes CRC*) //Reset
	
	B1_RES_LEN :BYTE := 29; (* Includes 2 Bytes START, 1 byte LEN + DATA + 2 Bytes CRC*)
	B2_RES_LEN :BYTE := 8; (* Includes 2 Bytes CRC*)
	B3_RES_LEN :BYTE := 8; (* Includes 2 Bytes CRC*)
	B4_RES_LEN :BYTE := 8; (* Includes 2 Bytes CRC*)
	B5_RES_LEN :BYTE := 10; (* Includes 2 Bytes CRC*)
	B8_RES_LEN :BYTE := 8; (* Includes 2 Bytes CRC*)
	CRC_CALC_LEN_ADJUST 	: BYTE 	:=	1; (* Include 2 btyes start, 1 byte len and remove 2 bytes of CRC*)
	TOTAL_MSG_LEN_ADJUST 	:BYTE 	:=	3; (* Include 2 bytes start and 1 byte of len*)
	FRAMING_HEADER			:BYTE	:=	3; (* Include 2 bytes start and 1 byte of len*)
	
	PLCPRJ_BUFFER_SIZE						: UDINT := 1000;(* Max. internal fifo/receiver buffer size *)

	PLCPRJ_CLIENT_SEND_CYCLE_TIME			: TIME := T#10S;
	PLCPRJ_RECEIVE_POLLING_TIME				: TIME := T#100MS;
	PLCPRJ_RECEIVE_TIMEOUT					: TIME := T#100S;

	(* Some project specific error codes *)
	PLCPRJ_ERROR_RECEIVE_TIMEOUT			: UDINT := 16#8101;(* Receive timeout *)
	PLCPRJ_ERROR_SENDFIFO_OVERFLOW			: UDINT := 16#8102;(* Send fifo overflow *)
	PLCPRJ_ERROR_RECFIFO_OVERFLOW			: UDINT := 16#8103;(* Receive fifo overflow *)
	PLCPRJ_ERROR_INVALID_FRAME_FORMAT		: UDINT := 16#8104;(* Invalid frame format/data *)
	
	MM_HLC_STATUS_POLLING					: TIME := T#60S;
	MM_PATH_STATUS_POLLING					: TIME := T#30S;
	MM_MOTOR_STATUS_POLLING					: TIME := T#60S;
	MM_VEHICLE_STATUS_POLLING				: TIME := T#1000MS;
	
	STATUS_REQ_TYPE_HLC		:BYTE :=16#0;
	STATUS_REQ_TYPE_NC		:BYTE :=16#1;
	STATUS_REQ_TYPE_Node	:BYTE :=16#2;
	STATUS_REQ_TYPE_Path	:BYTE :=16#3;
	STATUS_REQ_TYPE_Vehicle	:BYTE :=16#4;
	STATUS_REQ_TYPE_Motor	:BYTE :=16#5;
	
	HLC_STATE_INIT				:BYTE :=16#1;
	HLC_STATE_DEGRADED			:BYTE :=16#2;
	HLC_STATE_OPERATIONAL		:BYTE :=16#3;
	
	MAX_VEHICLES					:BYTE 	:= 20;
	
	MAX_STATIONS					:BYTE 	:= 13;
	
	LOAD_1_STA						:BYTE 	:= 1;
	LOAD_2_STA						:BYTE 	:= 2;
	LOAD_3_STA						:BYTE 	:= 3;
	LOAD_4_STA						:BYTE 	:= 4;
	STOP_BEFORE_BURNOFF_STA			:BYTE	:= 5;
	STOP_BEFORE_VISION_STA			:BYTE	:= 6;
	VISION_STA						:BYTE	:= 7;
	PISTON_STA						:BYTE	:= 8;
	CAP_STA							:BYTE	:= 9;
	IB_STOP_ROBOT_CLEAR_STA			:BYTE	:= 10;
	REJECT_ULOAD_STA				:BYTE	:= 11;	
	GOOD_UNLOAD_STA					:BYTE	:= 12;	
	OB_STOP_ROBOT_CLEAR_STA			:BYTE	:= 13;
	GOOD_UL_1_STA					:BYTE	:= 14;
	GOOD_UL_2_STA					:BYTE	:= 15;
	GOOD_UL_3_STA					:BYTE	:= 16;
	GOOD_UL_4_STA					:BYTE	:= 17;
	
	
	
	One_Meter						:REAL 	:= 1000; // One_Meter in mm
	Curved_Section_Length			:REAL 	:= 196.3495; //90 degree 125 mm radius
	Section_Gap						:REAL 	:= 2.2565; // gap in joints in mm
	Vehicle_Length					:REAL 	:= 100; //vehicle length
	Robot_Tool_Plate_Length			:REAL 	:= 480; //Tooling plate length on track in mm
	L1L2_Dist						:REAL 	:= 116.7384; //center to center distance between Load 1 and Load 2
	L2L3_Dist						:REAL 	:= 111.86160; //center to center distance between Load 2 and Load 3
	L3L4_Dist						:REAL 	:= 116.7384; //center to center distance between Load 3 and Load 4
	Min_Gap_Vehicle_Robot_Plate		:REAL 	:= 40; //minimum gap between robot tool plate end and begining of vehicle
    MinGapInterVehStationary        :REAL   := 20; //minimum gap between vehicles when stationary
	RejectStaAfterCurveSection      :REAL   := 50; //minimum gap between vehicles when stationary
 	
	(*
	LOAD_1_POS					     :REAL 	:= 0.8240;//0.8265;// 1.0262-0.2003;//(Curved_Section_Length +  Section_Gap + One_Meter - (L2L3_Dist/2) - L1L2_Dist)/1000; // in meters
	LOAD_2_POS					     :REAL 	:= 0.9414;//0.9435; //1.1442-0.2003;//(Curved_Section_Length +  Section_Gap + One_Meter - (L2L3_Dist/2))/1000; // in meters
	LOAD_3_POS					     :REAL 	:= 1.0539;//1.0549; //1.2562-0.2003;//(Curved_Section_Length +  Section_Gap + One_Meter + Section_Gap + (L2L3_Dist/2))/1000; // in meters
	LOAD_4_POS					     :REAL 	:= 1.17002;//1.1699; //1.3745-0.2003;//(Curved_Section_Length +  Section_Gap + One_Meter + Section_Gap + (L2L3_Dist/2) + L3L4_Dist)/1000; // in meters
	STOP_BEFORE_BURNOFF_POS		     :REAL	:= 1.5-0.2003;
	STOP_BEFORE_VISION_POS		     :REAL	:= 2.1-0.2003+0.076+0.100; //2.0757
	VISION_POS					     :REAL	:= 2.2005;//2.401725-0.2003;
	PISTON_POS					     :REAL	:= 2.8169;//3.0184-0.2003; //VISION_POS + (Curved_Section_Length+ Section_Gap + One_Meter - 574.09464)/1000;
	CAP_POS						     :REAL	:= 4.0628-0.2003;//VISION_POS + (Curved_Section_Length+ Section_Gap + One_Meter + Section_Gap + 454.84)/1000;
	IB_STOP_ROBOT_CLEAR_POS	 		 :REAL	:= VISION_POS + (Curved_Section_Length+ Section_Gap + One_Meter - 320)/1000;  // in meters;
	//REJECT_ULOAD_POS			     :REAL	:= VISION_POS + (Curved_Section_Length+ Section_Gap + One_Meter + Section_Gap + 816.74990)/1000;
	GOOD_UNLOAD_POS				     :REAL	:= 4.601;//4.5996;//4.602755;//4.8;	
	REJECT_ULOAD_POS			     :REAL	:= 0.0836; //0.2823-0.2003;// (Curved_Section_Length +  Section_Gap + RejectStaAfterCurveSection +25.4  )/1000; // in meters	
	OB_STOP_ROBOT_CLEAR_POS  		 :REAL	:= (One_Meter - 280)/1000; // in meters
	*)
	
	// New Positions for IMBAD4
	OB_STOP_ROBOT_CLEAR_POS  		 :REAL	:= 3.8000;
    LOAD_1_POS					     :REAL 	:= 3.95142;
	LOAD_2_POS					     :REAL 	:= 4.05175;
	LOAD_3_POS					     :REAL 	:= 4.1569;
	LOAD_4_POS					     :REAL 	:= 4.2569087;
	STOP_BEFORE_BURNOFF_POS		     :REAL	:= 4.4237; 
	STOP_BEFORE_VISION_POS		     :REAL	:= 0.010; 
	VISION_POS					     :REAL	:= 0.129; //0.13488; // 0.1266; nap 041919 
	PISTON_POS					     :REAL	:= 0.8661;
	IB_STOP_ROBOT_CLEAR_POS	 		 :REAL	:= 1.5; // not used any more
	CAP_POS						     :REAL	:= 2.26184759;
	GOOD_UNLOAD_POS				     :REAL	:= 3.1736 ; //never used 
	REJECT_ULOAD_POS			     :REAL	:= 3.170 ; 
	GOOD_UL_1_POS					 :REAL	:= 2.5888; //2.6460; //04/18/19 nap
	GOOD_UL_2_POS					 :REAL	:= 2.70843; //2.7138; //04/18/19 nap
	GOOD_UL_3_POS					 :REAL	:= 2.8381; //04/18/19 nap
	GOOD_UL_4_POS					 :REAL	:= 2.9055; //2.958; // 2.905346;  Changed by ALM 03/20/19
	
	
	
	AUTOBAGGER_HMI_STATE						:BYTE   := 1;
	CAP_STA_HMI_STATE							:BYTE	:= 2;
	CYCLE_CONTROL_HMI_STATE						:BYTE	:= 3;
	GOOD_UNLOAD_STA_HMI_STATE					:BYTE	:= 4;
	IB_STOP_ROBOT_CLEAR_STA_HMI_STATE			:BYTE	:= 5;
	IONIZER_HMI_STATE							:BYTE 	:= 6;
	LOAD_1_STA_HMI_STATE						:BYTE 	:= 7;
	LOAD_2_STA_HMI_STATE						:BYTE 	:= 8;
	LOAD_3_STA_HMI_STATE						:BYTE 	:= 9;
	LOAD_4_STA_HMI_STATE						:BYTE 	:= 10;
	MAIN_CONTROL_HMI_STATE						:BYTE	:= 11;
	OB_STOP_ROBOT_CLEAR_STA_HMI_STATE			:BYTE	:= 12;
	PISTON_STA_HMI_STATE						:BYTE	:= 13;
	PRIME_MOVER_HMI_STATE						:BYTE	:= 14;
	REJECT_ULOAD_STA_HMI_STATE					:BYTE	:= 15;
	ROBOT_STA_HMI_STATE							:BYTE 	:= 16;
	VISION_STA_HMI_STATE						:BYTE	:= 17;
	BURNOFF_STA_HMI_STATE						:BYTE	:= 18;
	GOOD_UL_1_STA_HMI_STATE						:BYTE	:= 19;
	GOOD_UL_2_STA_HMI_STATE						:BYTE	:= 20;
	GOOD_UL_3_STA_HMI_STATE						:BYTE	:= 21;
	GOOD_UL_4_STA_HMI_STATE						:BYTE	:= 22;
	
	
	
	
	
	
END_VAR

// ---- GVLs/PartsData.TcGVL
{attribute 'qualified_only'}
VAR_GLOBAL PERSISTENT 
	Status :ARRAY[1..MM_CONST.MAX_VEHICLES] OF PartDataType;
END_VAR

// ---- GVLs/Stations.TcGVL
{attribute 'qualified_only'}
VAR_GLOBAL
	fbMMClient		: MMClient ;(* Magnemotion Client (connection) instance *)
	fbMMSendMsg		: MM_MsgFormatter; (* Implements the Magnemotion TCP/IP Protocol and adds to TxFifo*)
	fbMMParseRes	: MM_MsgParser; (* Reads Magnemotion RxFifo and parses the data*)
	fbMMMonitor		: MMStatusMonitor; (* At periodic interval checks the status of MM elements*)
	fbCycleControl	: CycleControl; (* Controls Start/Stop Logic, I/O Locks, Reset and Homing Triggers*)
	fbPrimeMover	: PrimeMover; (* Will bring the Prime Move from a hard reset to all Vehicles in Init locations*)
	fbStationManager :StationManager; (* Triggers the right stations upon vehicle arrival*)
	fbVehicleManager : ARRAY[1..MM_CONST.MAX_VEHICLES] OF VehicleManager; (* Cmds Vehicles to Move, and monitors movement. Notifies arrival to Station Manager*)
	fbRoutePlanner	: RoutePlanner; (* Implements business logic of where to send the vehicles next after each station processing  *)
	fbLoad1Sta		: Load1Station;
	fbLoad2Sta		: Load2Station;
	fbLoad3Sta		: Load3Station;
	fbLoad4Sta		: Load4Station;
	fbOB_StopRobotSta		: OB_StopRobotClearStation;
	fbOB_StopBeforeVisionSta: OB_StopBeforeVisionStation;
	fbVisionSta				: VisionStation;
	fbPistonSta				: PistonInsertStation;
	fbIB_StopRobotSta		: IB_StopRobotClearStation;
	fbCapInsertSta			: CapInsertStation;
	fbGoodUnloadSta			: GoodUnloadStation;
	fbGoodULSta_1			: GoodULStation_1;
	fbGoodULSta_2			: GoodULStation_2;
	fbGoodULSta_3			: GoodULStation_3;
	fbGoodULSta_4			: GoodULStation_4;
	fbRejectSta				: RejectStation;
	fbBurnOffSta			: BurnOffStation;
	fbAutoBagger			: AutoBagger;
END_VAR

// ---- GVLs/STATUS.TcGVL
{attribute 'qualified_only'}
VAR_GLOBAL
	MMVehiclesStatus: ARRAY[1..MM_CONST.MAX_VEHICLES] OF ST_VehicleStatus;	(*Vehicle Status unpacked in data structure*)
	MMVehiclesStatusHMI: ARRAY[1..MM_CONST.MAX_VEHICLES] OF ST_VehicleStatusHMI;	(*Vehicle Status in Byte Array for ADS Comms*)
	StationsState : ARRAY[1..CONFIG.HMI_STATIONS_NUMB] OF INT;
	StationStauts : ARRAY[1..CONFIG.HMI_STATIONS_NUMB] OF INT;
	//StationStatusMsg: ARRAY[1..CONFIG.HMI_STATIONS_NUMB] OF STRING;
	StationInfoString: ARRAY[1..CONFIG.HMI_STATIONS_NUMB] OF STRING;
	IonizerStatusMsg:STRING;
	BurnOffStatusMsg:STRING;
	VisionStatusMsg:STRING;
	PistonStatusMsg:STRING;
	CapStatusMsg:STRING;
	GoodULStatusMsg:STRING;
	RejectStatusMsg:STRING;
	Load1StatusMsg:STRING;
	PrimeMoverStatusMsg:STRING;
	AutoBaggerStatusMsg:STRING;
	GoodUL_1_StatusMsg: STRING;
	GoodUL_2_StatusMsg: STRING;
	GoodUL_3_StatusMsg: STRING;
	GoodUL_4_StatusMsg: STRING;
	
	PartStatusHMI: ARRAY[1..MM_CONST.MAX_VEHICLES] OF INT;
	VisionStatusHMI: ARRAY[1..8] OF INT;
	BurnOffTemperature :DINT;
	BurnOffStatus : STRING;
	BaggerPrintCmd: BYTE;
	BurnOffIdle : BOOL := FALSE;
	
	ErrorMessage :STRING(80); 
	
END_VAR


// Part Present :0 Empty, 1 = Present
// Short Shot Pass : 0 Fail, Pass 1
// Camera2 Total Stain Count:
// Camera2 Total Stain Area
// Camera3 Total Stain Count:
// Camera3 Total Stain Area
// Camera4 Total Stain Count:
// Camera4 Total Stain Area

// ---- GVLs/VIS_CONST.TcGVL
{attribute 'qualified_only'}
VAR_GLOBAL
	Cmd_SwitchToRunMode : BYTE := 8;
	Cmd_ClearError		: BYTE := 13;
	Cmd_TriggerReset	: BYTE := 15;
	Cmd_ChangeProgram	: BYTE := 24;
	Cmd_ReadProgram 	: BYTE := 25;
END_VAR

// ---- POUs/MAIN.TcPOU
PROGRAM MAIN
VAR
	byCounter : BYTE:= 1;
	bInitialize :BOOL := TRUE;
	fbTick, fbIOLockedTick: TON;
	fbGetInputsFromFieldBus : GetInputsFromFieldBus;
	fbMapLockedOutputsFromHMI : MapLockedOutputsfromHMI;
	fbPrepareInputsForHMI : PrepareInputsDataStructureForHMI;
	fbPrepareOutputsForHMI : PrepareOutputsDataStructureForHMI;
	fbSetOutputsToFieldbus : SetOutputsToFieldbus;
	fbLotLogging : LotLogging;
	IOLocked : BOOL :=FALSE;	
	PrevIOLocked : BOOL := FALSE;
	fbEL6001	: FB_SerialCom;
	fbWritePersistentData 		: WritePersistentData;
	
END_VAR

Status.StationStauts[MM_CONST.IONIZER_HMI_STATE] := OverallStationStatus.eWaitingForParts;
//Set the Ionizer station to be blue on the HMI screen

//Logging 
LotsData.Lot.PLCVersion := '051319 v1.1.3'; //this goes into the HMI About Box. Lot is updated more frequently.

Logging.fbEventMsg();
Logging.fbEventMsgParams();
Logging.fbCurrTime();
P_TextModeWrite();(* This sample program opens and writes CSV file in text mode *)
P_TextModeWriteLot(); // this writes a lot report when end lot is written
fbLotLogging();
fbEL6001(TxBuffer:=GVL_IO.TxBufferEL, RxBuffer:= GVL_IO.RxBufferEL);
IF (bInitialize) THEN
	Logging.fbEventMsg.SendEventMsg(MsgClass := TCEVENTCLASS_STATEINFO, EventID:= Logging.IDMain_InitBegin , SourceID:= Logging.SrcMainPOU);
	bInitialize := FALSE;
END_IF

// Magnemotion Communication 
Stations.fbMMClient();
// Only Accept Cmds to Magnemotion and Parse Responses from Magnemotion HLC when socket is connected.
// To DO: Document the software architecture and timeout/error handling
IF (Stations.fbMMClient.eState = eSOCKET_CONNECTED) THEN
	Stations.fbMMSendMsg(fbTx:=Stations.fbMMClient.fbTx, fbLog := Stations.fbMMClient.fbLog);
	Stations.fbMMParseRes(fbRx:=Stations.fbMMClient.fbRx, fbLog := Stations.fbMMClient.fbLog);
	Stations.fbMMMonitor();	
ELSE ;	
END_IF	


// Beckhoff Run time (XAR) will fetch all the fieldbus data and map to GVL_IO variables whereever mapping is directly addressable 
// For the Inputs where we have to program the linking of I/O variables to the fieldbus data, we need to execute this routine once 
// every cycle
fbGetInputsFromFieldBus(); //Mapping of bytes into PLC variables, where such mapping is not available in I/O linking directly

// Machine is E-Stopped
// Each station will set its Current State and Next State to Unknown condition when Machine is E-Stopped
// After Reset condition we need the operator to hit the start button and the air to be at correct pressure for each station to proceed
IF (GVL_IO.MachineEStopped) THEN	
;
ELSE
//	GVL_IO.VS_YBarrelLED := TRUE; 	// to do, change this so that the logic is handled by the respective station 
END_IF


IOLocked := (GVL_IO.IOLockedFromHMI <>0);
IF (PrevIOLocked AND NOT IOLocked) THEN
	//send all stations to Unknown State when we move from IO Locked state to IO Unlocked State.
	ResetAllStations();	
END_IF
PrevIOLocked := IOLocked;

IF (IOLocked) THEN  //Don't execute and PLC logic to control outputs.. however execute the temperature control logic.
	fbMapLockedOutputsFromHMI(); // get outputs state from HMI.     
//	GVL_IO.MM_YEnableMagneMotion := FALSE; // Unclear if this is needed, but for now we are disabling Prime Mover when I/O is locked
    //Send Timer based Messages to the Operator HMI
    fbIOLockedTick(IN:=TRUE, PT:= T#5M); //To Add, add CPU monitoring parameters to report out, temperature, memory etc.
	IF (fbIOLockedTick.Q) THEN
		Logging.fbEventMsg.SendEventMsg(MsgClass := TCEVENTCLASS_WARNING,EventID:= Logging.IDMain_Tick , SourceID:= Logging.SrcMainPOU);
		fbIOLockedTick(IN:=FALSE);
	END_IF (* IO Tick Timer Event*)
ELSE  // Run normally without IO being locked
    //Tick for Stations --- these stations do not get called when I/O is locked. They will return to Unkonwn state after I/O is again unlocked from a locked state
	Stations.fbLoad1Sta();  // Load 1 Station which also handles Yushin Communication and Load Station Cyclinders
	Stations.fbLoad2Sta();  // Load 2 
	Stations.fbLoad3Sta();  // Load 3 
	Stations.fbLoad4Sta();  // Load 4
	Stations.fbVisionSta(); // Vision Station			 	
	Stations.fbPistonSta();  // Piston Insert 	
	Stations.fbCapInsertSta();	 //Cap Insert 
	//Stations.fbGoodUnloadSta();  // Good Unload 			 
	Stations.fbRejectSta();	 //Reject Station			
	Stations.fbAutoBagger();
	Stations.fbGoodULSta_1();
	Stations.fbGoodULSta_2();
	Stations.fbGoodULSta_3();
	Stations.fbGoodULSta_4();
END_IF (* If IO Locked*)
// Run all the other stations at all times 
// Cycle management and interlocks
Stations.fbIB_StopRobotSta();		// Stop for Yushin Load plate inbound side
Stations.fbOB_StopRobotSta(); // Stop for Yushin Load Plate outbound side
Stations.fbOB_StopBeforeVisionSta(); // Stop before Vision station
Stations.fbCycleControl();
Stations.fbStationManager();  // Allows Vehicle Manager to trigger stations after vehicle arrives under a station
Stations.fbRoutePlanner();  // This allows Stations to Inform Vehicle Manager processing is complete, adds logic for route planning
	
Stations.fbPrimeMover(); // Primve Mover
FOR byCounter := 1 TO MM_CONST.MAX_VEHICLES BY 1 DO
			Stations.fbVehicleManager[byCounter](VehicleID := byCounter);  // Vehicle Manager
END_FOR
Stations.fbBurnOffSta(); // Burn off station - handles PID control and cools of burn off this needs to run regardless of I/O Lock

fbPrepareInputsForHMI(); // Send copy of Input State to the PC HMI Byte Array -- to refresh the HMI ( Note that HMI requests the refresh)
fbPrepareOutputsForHMI(); //Send Copy of the Output State to the PC HMI Byte Array -- to refresh the HMI (Note that HMI requests the refresh)

// Beckhoff Run time (XAR) will write all the fieldbus data and map to GVL_IO variables whereever mapping is directly addressable 
// For the Output where we have to program the linking of I/O variables to the fieldbus data, we need to execute this routine once 
// every cycle

fbSetOutputstoFieldbus(); // //Mapping of bytes into Fieldbus variables, where such mapping is not available in I/O linking directly


// A tick message to the operator logging screen 

fbTick(IN:=TRUE, PT:= T#60S); //To Add, add CPU monitoring parameters to report out, temperature, memory etc.
IF (fbTick.Q) THEN
	Logging.fbEventMsg.SendEventMsg(MsgClass := TCEVENTCLASS_STATEINFO, EventID:= Logging.IDMain_Tick , SourceID:= Logging.SrcMainPOU);
	fbWritePersistentData(NETID:='', PORT:=851, START:=TRUE, TMOUT:=T#1S );
	fbTick(IN:=FALSE);
ELSE
	fbWritePersistentData(NETID:='', PORT:=851, START:=FALSE, TMOUT:=T#1S );
END_IF
Status.StationsState[MM_CONST.MAIN_CONTROL_HMI_STATE] := BOOL_TO_INT(IOLocked)+501;

METHOD PUBLIC ResetAllStations : BOOL
VAR_INPUT
END_VAR
Stations.fbLoad1Sta.ResetState();
Stations.fbLoad2Sta.ResetState();
Stations.fbLoad3Sta.ResetState();
Stations.fbLoad4Sta.ResetState();
//Stations.fbVisionSta();  // TO DO			
Stations.fbPistonSta.ResetState();
//Stations.fbIB_StopRobotSta();		
Stations.fbCapInsertSta.ResetState();
//Stations.fbGoodUnloadSta.ResetState();	
Stations.fbGoodULSta_1.ResetState();
Stations.fbGoodULSta_2.ResetState();
Stations.fbGoodULSta_3.ResetState();
Stations.fbGoodULSta_4.ResetState();	
Stations.fbRejectSta.ResetState();
//Stations.fbOB_StopRobotSta();
//Stations.fbOB_StopBeforeVisionSta();
//Stations.fbBurnOffSta();   TO DO
END_METHOD

END_PROGRAM

// ---- POUs/FrameworkPOUs/GetInputsFromFieldBus.TcPOU
// Fill up the appropriate IO from the inputs coming from the field which are not directly addressable in the linking of variables
FUNCTION_BLOCK FINAL GetInputsFromFieldBus
VAR_INPUT
END_VAR
VAR_OUTPUT
END_VAR
VAR
	SMCMtrPosRawByte3 : DWORD;
	SMCMtrPosRawByte2 : DWORD;
	SMCMtrPosRawByte1 : DWORD;
	SMCMtrPosRawByte0 : DWORD;
	SMCMtrPosRaw	  : DINT;	
	
	RawByte3: DWORD;
	RawByte2: DWORD;
	RawByte1: DWORD;
	RawByte0: DWORD;
	RawDWORD : DWORD;
	UL: INT;
END_VAR

GVL_IO.PI_XMtrOUT0 := GVL_IO.SMC_LEY_XUINT0.0;
GVL_IO.PI_XMtrOUT1 := GVL_IO.SMC_LEY_XUINT0.1;  
GVL_IO.PI_XMtrOUT2 := GVL_IO.SMC_LEY_XUINT0.2; 
GVL_IO.PI_XMtrOUT3 := GVL_IO.SMC_LEY_XUINT0.3; 
GVL_IO.PI_XMtrOUT4 := GVL_IO.SMC_LEY_XUINT0.4; 
GVL_IO.PI_XMtrOUT5 := GVL_IO.SMC_LEY_XUINT0.5; 

GVL_IO.PI_XMtrBusy 			:= GVL_IO.SMC_LEY_XUINT0.8;
GVL_IO.PI_XMtrServoEnabled 	:= GVL_IO.SMC_LEY_XUINT0.9;
GVL_IO.PI_XMtrServoHomed 	:= GVL_IO.SMC_LEY_XUINT0.10; 
GVL_IO.PI_XMtrMoveCompl 	:= GVL_IO.SMC_LEY_XUINT0.11;
GVL_IO.PI_XMtrEStopped 		:= GVL_IO.SMC_LEY_XUINT0.12;
GVL_IO.PI_XMtrAlarm 		:= GVL_IO.SMC_LEY_XUINT0.13;
GVL_IO.PI_XMtrReady			:= GVL_IO.SMC_LEY_XUINT1.4;

GVL_IO.PI_XMtrCurrPos := DINT_TO_REAL(GVL_IO.SMC_LEY_XCurrMtrPos)/100;

//GVL_IO.MC_NotEStopped := GVL_IO.MC_XAirPressureOK; // overriding this until MOV is in place
GVL_IO.MachineEStopped := NOT GVL_IO.MC_NotEStopped; // Better code readability 

GVL_IO.UL_XPP_DriveEnabled := GVL_IO.UL_XPP_Byte4.0;
GVL_IO.UL_XPP_StopActive := GVL_IO.UL_XPP_Byte4.1;
GVL_IO.UL_XPP_ReferenceOK := GVL_IO.UL_XPP_Byte4.2;
GVL_IO.UL_XPP_ReadyToStart := GVL_IO.UL_XPP_Byte4.3;
GVL_IO.UL_XPP_Alarm := GVL_IO.UL_XPP_Byte4.4;
GVL_IO.UL_XPP_A1OUT := GVL_IO.UL_XPP_Byte4.5;
GVL_IO.UL_XPP_A2OUT := GVL_IO.UL_XPP_Byte4.6;
GVL_IO.UL_XPP_A3OUT := GVL_IO.UL_XPP_Byte4.7;
GVL_IO.UL_XPP_LubeLevel := GVL_IO.UL_XPP_Byte5.0;

// Vision 

GVL_IO.VS_XCmdCmpl := GVL_IO.VS_XByte0.0;
GVL_IO.VS_XCmdErr  := GVL_IO.VS_XByte0.1;
GVL_IO.VS_XCmdReady := GVL_IO.VS_XByte0.2;
GVL_IO.VS_XResultReady := GVL_IO.VS_XByte0.3;
GVL_IO.VS_XResultOR := GVL_IO.VS_XByte0.4;
GVL_IO.VS_XCmdResult := GVL_IO.VS_XByte20;
GVL_IO.VS_XCmdData1 := GVL_IO.VS_XByte24;
GVL_IO.VS_XCmdData2 := GVL_IO.VS_XByte28;

GVL_IO.VS_XReady1 := GVL_IO.VS_XByte1.0;
GVL_IO.VS_XReady2 := GVL_IO.VS_XByte1.1;
GVL_IO.VS_XReady3 := GVL_IO.VS_XByte1.2;
GVL_IO.VS_XReady4 := GVL_IO.VS_XByte1.3;

GVL_IO.VS_XAck1 := GVL_IO.VS_XByte2.0;
GVL_IO.VS_XAck2 := GVL_IO.VS_XByte2.1;
GVL_IO.VS_XAck3 := GVL_IO.VS_XByte2.2;
GVL_IO.VS_XAck4 := GVL_IO.VS_XByte2.3;

GVL_IO.VS_XBusy :=  GVL_IO.VS_XByte3.0;
GVL_IO.VS_XError := GVL_IO.VS_XByte3.1;
GVL_IO.VS_XRun :=   GVL_IO.VS_XByte3.3;

GVL_IO.VS_XAllCamJudgeVal := GVL_IO.VS_XByte4.0;
GVL_IO.VS_XCam1JudgeVal := GVL_IO.VS_XByte4.1;
GVL_IO.VS_XCam2JudgeVal := GVL_IO.VS_XByte4.2;
GVL_IO.VS_XCam3JudgeVal := GVL_IO.VS_XByte4.3;
GVL_IO.VS_XCam4JudgeVal := GVL_IO.VS_XByte4.4;
GVL_IO.VS_XPartEmpty :=    GVL_IO.VS_XByte4.5;

GVL_IO.VS_XMaxIndividualStainArea := DINT_TO_REAL(GetRawDword(Byte0 := GVL_IO.VS_XByte48, Byte1:= GVL_IO.VS_XByte49, Byte2:= GVL_IO.VS_XByte50, Byte3:= GVL_IO.VS_XByte51))/ 1000;
GVL_IO.VS_XMinIndividualStainArea := DINT_TO_REAL(GetRawDword(Byte0 := GVL_IO.VS_XByte52, Byte1:= GVL_IO.VS_XByte53, Byte2:= GVL_IO.VS_XByte54, Byte3:= GVL_IO.VS_XByte55))/ 1000;
GVL_IO.VS_XModifiedStainArea	:= DINT_TO_REAL(GetRawDword(Byte0 := GVL_IO.VS_XByte56, Byte1:= GVL_IO.VS_XByte57, Byte2:= GVL_IO.VS_XByte58, Byte3:= GVL_IO.VS_XByte59))/ 1000;
GVL_IO.VS_XModifiedMaxStain		:= DINT_TO_REAL(GetRawDword(Byte0 := GVL_IO.VS_XByte60, Byte1:= GVL_IO.VS_XByte61, Byte2:= GVL_IO.VS_XByte62, Byte3:= GVL_IO.VS_XByte63))/ 1000;
GVL_IO.VS_XYPosCam1 			:= DINT_TO_REAL(GetRawDword(Byte0 := GVL_IO.VS_XByte64, Byte1:= GVL_IO.VS_XByte65, Byte2:= GVL_IO.VS_XByte66, Byte3:= GVL_IO.VS_XByte67))/ 1000;

GVL_IO.VS_XUpperFlawAreaCam2	:= GetRawDword(Byte0 := GVL_IO.VS_XByte68, Byte1:= GVL_IO.VS_XByte69, Byte2:= GVL_IO.VS_XByte70, Byte3:= GVL_IO.VS_XByte71);
GVL_IO.VS_XLowerFlawAreaCam2	:= GetRawDword(Byte0 := GVL_IO.VS_XByte72, Byte1:= GVL_IO.VS_XByte73, Byte2:= GVL_IO.VS_XByte74, Byte3:= GVL_IO.VS_XByte75);
GVL_IO.VS_XUpperFlawCountCam2	:= GetRawDword(Byte0 := GVL_IO.VS_XByte76, Byte1:= GVL_IO.VS_XByte77, Byte2:= GVL_IO.VS_XByte78, Byte3:= GVL_IO.VS_XByte79);
GVL_IO.VS_XLowerFlawCountCam2	:= GetRawDword(Byte0 := GVL_IO.VS_XByte80, Byte1:= GVL_IO.VS_XByte81, Byte2:= GVL_IO.VS_XByte82, Byte3:= GVL_IO.VS_XByte83);

GVL_IO.VS_XUpperFlawAreaCam3	:= GetRawDword(Byte0 := GVL_IO.VS_XByte88, Byte1:= GVL_IO.VS_XByte89, Byte2:= GVL_IO.VS_XByte90, Byte3:= GVL_IO.VS_XByte91);
GVL_IO.VS_XLowerFlawAreaCam3	:= GetRawDword(Byte0 := GVL_IO.VS_XByte92, Byte1:= GVL_IO.VS_XByte93, Byte2:= GVL_IO.VS_XByte94, Byte3:= GVL_IO.VS_XByte95);
GVL_IO.VS_XUpperFlawCountCam3	:= GetRawDword(Byte0 := GVL_IO.VS_XByte96, Byte1:= GVL_IO.VS_XByte97, Byte2:= GVL_IO.VS_XByte98, Byte3:= GVL_IO.VS_XByte99);
GVL_IO.VS_XLowerFlawCountCam3	:= GetRawDword(Byte0 := GVL_IO.VS_XByte100, Byte1:= GVL_IO.VS_XByte101, Byte2:= GVL_IO.VS_XByte102, Byte3:= GVL_IO.VS_XByte103);

GVL_IO.VS_XUpperFlawAreaCam4	:= GetRawDword(Byte0 := GVL_IO.VS_XByte108, Byte1:= GVL_IO.VS_XByte109, Byte2:= GVL_IO.VS_XByte110, Byte3:= GVL_IO.VS_XByte111);
GVL_IO.VS_XLowerFlawAreaCam4	:= GetRawDword(Byte0 := GVL_IO.VS_XByte112, Byte1:= GVL_IO.VS_XByte113, Byte2:= GVL_IO.VS_XByte114, Byte3:= GVL_IO.VS_XByte115);
GVL_IO.VS_XUpperFlawCountCam4	:= GetRawDword(Byte0 := GVL_IO.VS_XByte116, Byte1:= GVL_IO.VS_XByte117, Byte2:= GVL_IO.VS_XByte118, Byte3:= GVL_IO.VS_XByte119);
GVL_IO.VS_XLowerFlawCountCam4	:= GetRawDword(Byte0 := GVL_IO.VS_XByte120, Byte1:= GVL_IO.VS_XByte121, Byte2:= GVL_IO.VS_XByte122, Byte3:= GVL_IO.VS_XByte123);


// Some HMI ADS related data

IF (LotsData.Lot.BarrelSizeInt = 55) THEN
	LotsData.Lot.BarrelSize := eBarrelType.Size55cc;
ELSIF (LotsData.Lot.BarrelSizeInt = 30) THEN
	LotsData.Lot.BarrelSize := eBarrelType.Size30cc;
ELSIF (LotsData.Lot.BarrelSizeInt = 10) THEN
	LotsData.Lot.BarrelSize := eBarrelType.Size10cc;
ELSIF (LotsData.Lot.BarrelSizeInt = 5) THEN
	LotsData.Lot.BarrelSize := eBarrelType.Size5cc;
ELSIF (LotsData.Lot.BarrelSizeInt = 3) THEN
	LotsData.Lot.BarrelSize := eBarrelType.Size3cc;
ELSE
	LotsData.Lot.BarrelSize := eBarrelType.Size55cc;
END_IF

IF (LotsData.Lot.VisionStationRunSelectInt = 0) THEN
	LotsData.Lot.VisionStationRunSelect := eVisionEnableState.Disabled;
ELSIF (LotsData.Lot.VisionStationRunSelectInt = 1) THEN
	LotsData.Lot.VisionStationRunSelect := eVisionEnableState.Enabled;
ELSIF (LotsData.Lot.VisionStationRunSelectInt = 2) THEN
	LotsData.Lot.VisionStationRunSelect := eVisionEnableState.DataCollectOnly;
END_IF

METHOD PUBLIC GetRawDword : DINT
VAR_INPUT
	Byte0: DWORD;
	Byte1: DWORD;
	Byte2: DWORD;
	Byte3: DWORD;
END_VAR
GetRawDword := SHL(Byte3,24) OR SHL(Byte2,16) OR SHL(Byte1,8) OR Byte0;
END_METHOD

END_FUNCTION_BLOCK

// ---- POUs/FrameworkPOUs/MapLockedOutputsfromHMI.TcPOU
// Get the outputs directly from the HMI and map them to internal PLC IO variables. During this condition, all of the PLC Logic is bypassed
// Coming out of this routine, we should set the states of the stations to UnKnown.
FUNCTION_BLOCK PUBLIC MapLockedOutputsfromHMI
VAR_INPUT
END_VAR
VAR_OUTPUT
END_VAR
VAR
END_VAR

GVL_IO.LD_YPalletHoldDownRetractEngage  := BYTE_TO_BOOL(GVL_IO.OutputsFromHMI[1]);
GVL_IO.LD_YPalletHoldDownExtendHome := BYTE_TO_BOOL(GVL_IO.OutputsFromHMI[2]);
GVL_IO.LD_YPalletReleaseExtend   := BYTE_TO_BOOL(GVL_IO.OutputsFromHMI[3]);
GVL_IO.LD_YPalletReleaseRetract  := BYTE_TO_BOOL(GVL_IO.OutputsFromHMI[4]);
GVL_IO.LD_YPalletCloseExtend  := BYTE_TO_BOOL(GVL_IO.OutputsFromHMI[8]);
GVL_IO.LD_YPalletCloseRetract := BYTE_TO_BOOL(GVL_IO.OutputsFromHMI[9]);

// Yushin Robot Interface Outputs

GVL_IO.YU_YOkToLoad            := BYTE_TO_BOOL(GVL_IO.OutputsFromHMI[5]);
GVL_IO.YU_YAckPartsHeld        := BYTE_TO_BOOL(GVL_IO.OutputsFromHMI[6]);
GVL_IO.YU_YIMBADIsOK       	   := BYTE_TO_BOOL(GVL_IO.OutputsFromHMI[10]);


//Ionizer Outputs

GVL_IO.IZ_YInterrupt 			:= BYTE_TO_BOOL(GVL_IO.OutputsFromHMI[7]); 
//GVL_IO.IZ_YIonizerAirON 		:= BYTE_TO_BOOL(GVL_IO.OutputsFromHMI[8]);
//GVL_IO.IZ_YIonizerAirOFF 		:= BYTE_TO_BOOL(GVL_IO.OutputsFromHMI[9]);  

// Vision
GVL_IO.VS_YBarrelLED			:= BYTE_TO_BOOL(GVL_IO.OutputsFromHMI[21]);
GVL_IO.VS_YCmdRequest           := BYTE_TO_BOOL(GVL_IO.OutputsFromHMI[22]); 
GVL_IO.VS_YResultAck            := BYTE_TO_BOOL(GVL_IO.OutputsFromHMI[23]);
GVL_IO.VS_YErrorReset           := BYTE_TO_BOOL(GVL_IO.OutputsFromHMI[24]);
GVL_IO.VS_YTrigger1             := BYTE_TO_BOOL(GVL_IO.OutputsFromHMI[25]);
GVL_IO.VS_YTrigger2             := BYTE_TO_BOOL(GVL_IO.OutputsFromHMI[26]);
GVL_IO.VS_YTrigger3             := BYTE_TO_BOOL(GVL_IO.OutputsFromHMI[27]);
GVL_IO.VS_YTrigger4             := BYTE_TO_BOOL(GVL_IO.OutputsFromHMI[28]);






// Piston Insert 
GVL_IO.PI_YPalletHoldDownExtend  := BYTE_TO_BOOL(GVL_IO.OutputsFromHMI[31]);
GVL_IO.PI_YPalletHoldDownRetract := BYTE_TO_BOOL(GVL_IO.OutputsFromHMI[32]);
GVL_IO.PI_YEscapementToBowl      := BYTE_TO_BOOL(GVL_IO.OutputsFromHMI[33]);
GVL_IO.PI_YEscapementToWork      := BYTE_TO_BOOL(GVL_IO.OutputsFromHMI[34]);
GVL_IO.PI_YBarrelBackupExtend    := BYTE_TO_BOOL(GVL_IO.OutputsFromHMI[35]);
GVL_IO.PI_YBarrelBackupRetract   := BYTE_TO_BOOL(GVL_IO.OutputsFromHMI[36]);

GVL_IO.PI_YMtrStepSelectIN0		 := BYTE_TO_BOOL(GVL_IO.OutputsFromHMI[40]);
GVL_IO.PI_YMtrStepSelectIN1		 := BYTE_TO_BOOL(GVL_IO.OutputsFromHMI[41]);
GVL_IO.PI_YMtrStepSelectIN2      := BYTE_TO_BOOL(GVL_IO.OutputsFromHMI[42]);
GVL_IO.PI_YMtrHoldMove		     := BYTE_TO_BOOL(GVL_IO.OutputsFromHMI[43]);
GVL_IO.PI_YMtrSetEnable     	 := BYTE_TO_BOOL(GVL_IO.OutputsFromHMI[44]);
GVL_IO.PI_YMtrDriveStepTrigger   := BYTE_TO_BOOL(GVL_IO.OutputsFromHMI[45]);
GVL_IO.PI_YMtrReset			     := BYTE_TO_BOOL(GVL_IO.OutputsFromHMI[46]);
GVL_IO.PI_YMtrGoHome			 := BYTE_TO_BOOL(GVL_IO.OutputsFromHMI[47]);
GVL_IO.PI_YMtrJogNeg			 := BYTE_TO_BOOL(GVL_IO.OutputsFromHMI[48]);
GVL_IO.PI_YMtrJogPos			 := BYTE_TO_BOOL(GVL_IO.OutputsFromHMI[49]);
GVL_IO.PI_YMtrSwitchJogInch		 := BYTE_TO_BOOL(GVL_IO.OutputsFromHMI[50]);


// Cap Insert 

GVL_IO.CP_YCapSlideExtend 				:= BYTE_TO_BOOL(GVL_IO.OutputsFromHMI[57]);
GVL_IO.CP_YCapSlideRetract 				:= BYTE_TO_BOOL(GVL_IO.OutputsFromHMI[58]);
GVL_IO.CP_YPalletHoldDownExtend 		:= BYTE_TO_BOOL(GVL_IO.OutputsFromHMI[59]);
GVL_IO.CP_YPalletHoldDownRetract 		:= BYTE_TO_BOOL(GVL_IO.OutputsFromHMI[60]);


// Good Unload Outputs
GVL_IO.UL_1_YPalletHoldDownExtend_Home        := BYTE_TO_BOOL(GVL_IO.OutputsFromHMI[71]);
GVL_IO.UL_1_YPalletHoldDownRetract_Engage     := BYTE_TO_BOOL(GVL_IO.OutputsFromHMI[72]);
GVL_IO.UL_2_YPalletHoldDownExtend_Home        := BYTE_TO_BOOL(GVL_IO.OutputsFromHMI[73]);
GVL_IO.UL_2_YPalletHoldDownRetract_Engage     := BYTE_TO_BOOL(GVL_IO.OutputsFromHMI[74]);
GVL_IO.UL_3_YPalletHoldDownExtend_Home        := BYTE_TO_BOOL(GVL_IO.OutputsFromHMI[75]);
GVL_IO.UL_3_YPalletHoldDownRetract_Engage     := BYTE_TO_BOOL(GVL_IO.OutputsFromHMI[76]);
GVL_IO.UL_4_YPalletHoldDownExtend_Home        := BYTE_TO_BOOL(GVL_IO.OutputsFromHMI[77]);
GVL_IO.UL_4_YPalletHoldDownRetract_Engage     := BYTE_TO_BOOL(GVL_IO.OutputsFromHMI[78]);
                                                              
GVL_IO.UL_1_YRejectPushExtend                 := BYTE_TO_BOOL(GVL_IO.OutputsFromHMI[79]);
GVL_IO.UL_2_YRejectPushExtend                 := BYTE_TO_BOOL(GVL_IO.OutputsFromHMI[80]);
GVL_IO.UL_3_YRejectPushExtend                 := BYTE_TO_BOOL(GVL_IO.OutputsFromHMI[81]);
GVL_IO.UL_4_YRejectPushExtend                 := BYTE_TO_BOOL(GVL_IO.OutputsFromHMI[82]);

GVL_IO.UL_1_YRejectPushRetract                 := BYTE_TO_BOOL(GVL_IO.OutputsFromHMI[83]);
GVL_IO.UL_2_YRejectPushRetract	               := BYTE_TO_BOOL(GVL_IO.OutputsFromHMI[84]);
GVL_IO.UL_3_YRejectPushRetract                 := BYTE_TO_BOOL(GVL_IO.OutputsFromHMI[85]);
GVL_IO.UL_4_YRejectPushRetract                 := BYTE_TO_BOOL(GVL_IO.OutputsFromHMI[86]);
                                                                                                           

